LIN {X -0.181,Y -585.120,Z 1414.971,A 0.000,B 0.000,C 90.000,E1 30.797} C_DIS
LIN {X -0.267,Y -582.013,Z 1414.967,A 0.000,B 0.000,C 90.000,E1 30.001} C_DIS
LIN {X -0.018,Y -577.192,Z 1414.961,A 0.000,B 0.000,C 90.000,E1 28.899} C_DIS
LIN {X -0.191,Y -573.056,Z 1414.956,A 0.000,B 0.000,C 90.000,E1 28.103} C_DIS
LIN {X 0.092,Y -568.645,Z 1414.952,A 0.000,B 0.000,C 90.000,E1 27.257} C_DIS
LIN {X 0.067,Y -563.902,Z 1414.947,A 0.000,B 0.000,C 90.000,E1 26.437} C_DIS
LIN {X -0.163,Y -559.631,Z 1414.943,A 0.000,B 0.000,C 90.000,E1 25.771} C_DIS
LIN {X 0.221,Y -554.124,Z 1414.938,A 0.000,B 0.000,C 90.000,E1 24.899} C_DIS
LIN {X -0.222,Y -550.199,Z 1414.935,A 0.000,B 0.000,C 90.000,E1 24.387} C_DIS
LIN {X 0.061,Y -543.773,Z 1414.931,A 0.000,B 0.000,C 90.000,E1 23.515} C_DIS
LIN {X -0.088,Y -538.027,Z 1414.927,A 0.000,B 0.000,C 90.000,E1 22.823} C_DIS
LIN {X -0.189,Y -529.500,Z 1414.921,A 0.000,B 0.000,C 90.000,E1 21.844} C_DIS
LIN {X -0.178,Y -524.439,Z 1414.918,A 0.000,B 0.000,C 90.000,E1 21.280} C_DIS
LIN {X -0.246,Y -515.235,Z 1414.913,A 0.000,B 0.000,C 90.000,E1 20.301} C_DIS
LIN {X 0.169,Y -504.397,Z 1414.906,A 0.000,B 0.000,C 90.000,E1 19.141} C_DIS
LIN {X 0.226,Y -493.820,Z 1414.901,A 0.000,B 0.000,C 90.000,E1 18.055} C_DIS
LIN {X -0.129,Y -476.219,Z 1414.890,A 0.000,B 0.000,C 90.000,E1 16.260} C_DIS
LIN {X -0.019,Y -462.613,Z 1414.882,A 0.000,B 0.000,C 90.000,E1 14.773} C_DIS
LIN {X -0.025,Y -453.110,Z 1414.876,A 0.000,B 0.000,C 90.000,E1 13.716} C_DIS
LIN {X 0.077,Y -438.094,Z 1414.867,A 0.000,B 0.000,C 90.000,E1 12.007} C_DIS
LIN {X 0.034,Y -420.561,Z 1414.855,A 0.000,B 0.000,C 90.000,E1 9.905} C_DIS
LIN {X -0.065,Y -404.897,Z 1414.844,A 0.000,B 0.000,C 90.000,E1 7.871} C_DIS
LIN {X 0.079,Y -389.907,Z 1414.832,A 0.000,B 0.000,C 90.000,E1 5.796} C_DIS
LIN {X 0.032,Y -388.630,Z 1414.831,A 0.000,B 0.000,C 90.000,E1 5.625} C_DIS
LIN {X -0.056,Y -384.934,Z 1414.828,A 0.000,B 0.000,C 90.000,E1 4.992} C_DIS
LIN {X 0.034,Y -384.710,Z 1414.827,A 0.000,B 0.000,C 90.000,E1 4.878} C_DIS
LIN {X -0.003,Y -384.706,Z 1414.827,A 0.000,B 0.000,C 90.000,E1 4.878} C_DIS
LIN {X 0.112,Y -386.090,Z 1414.825,A 0.000,B 0.000,C 90.000,E1 4.473} C_DIS
LIN {X 0.057,Y -386.910,Z 1414.824,A 0.000,B 0.000,C 90.000,E1 4.302} C_DIS
LIN {X -0.075,Y -390.185,Z 1414.821,A 0.000,B 0.000,C 90.000,E1 3.784} C_DIS
LIN {X 0.181,Y -393.301,Z 1414.818,A 0.000,B 0.000,C 90.000,E1 3.212} C_DIS
LIN {X 0.160,Y -394.127,Z 1414.817,A 0.000,B 0.000,C 90.000,E1 3.037} C_DIS
LIN {X 0.084,Y -394.922,Z 1414.815,A 0.000,B 0.000,C 90.000,E1 2.694} C_DIS
LIN {X 0.145,Y -394.640,Z 1414.814,A 0.000,B 0.000,C 90.000,E1 2.579} C_DIS
LIN {X -0.179,Y -394.309,Z 1414.814,A 0.000,B 0.000,C 90.000,E1 2.579} C_DIS
LIN {X 0.177,Y -393.144,Z 1414.814,A 0.000,B 0.000,C 90.000,E1 2.465} C_DIS
LIN {X 0.102,Y -392.450,Z 1414.814,A 0.000,B 0.000,C 90.000,E1 2.465} C_DIS
LIN {X 0.060,Y -361.246,Z 1414.814,A 0.000,B 0.000,C 90.000,E1 2.465} C_DIS
LIN {X -0.064,Y -360.858,Z 1414.801,A 0.000,B 0.000,C 90.000,E1 0.115} C_DIS
LIN {X -0.053,Y -359.426,Z 1414.770,A 0.000,B 0.000,C 90.000,E1 354.546} C_DIS
LIN {X 0.070,Y -358.890,Z 1414.759,A 0.000,B 0.000,C 90.000,E1 352.648} C_DIS
LIN {X -0.020,Y -359.563,Z 1414.726,A 0.000,B 0.000,C 90.000,E1 346.645} C_DIS
LIN {X 0.001,Y -361.801,Z 1414.684,A 0.000,B 0.000,C 90.000,E1 339.135} C_DIS
LIN {X -0.154,Y -362.053,Z 1414.680,A 0.000,B 0.000,C 90.000,E1 338.411} C_DIS
LIN {X 0.189,Y -365.980,Z 1414.643,A 0.000,B 0.000,C 90.000,E1 331.641} C_DIS
LIN {X 0.029,Y -366.387,Z 1414.639,A 0.000,B 0.000,C 90.000,E1 330.923} C_DIS
LIN {X -0.031,Y -371.355,Z 1414.604,A 0.000,B 0.000,C 90.000,E1 324.642} C_DIS
LIN {X -0.043,Y -371.766,Z 1414.602,A 0.000,B 0.000,C 90.000,E1 324.276} C_DIS
LIN {X 0.013,Y -377.358,Z 1414.567,A 0.000,B 0.000,C 90.000,E1 318.038} C_DIS
LIN {X 0.012,Y -378.235,Z 1414.563,A 0.000,B 0.000,C 90.000,E1 317.310} C_DIS
LIN {X 0.002,Y -383.940,Z 1414.531,A 0.000,B 0.000,C 90.000,E1 311.515} C_DIS
LIN {X 0.088,Y -384.893,Z 1414.527,A 0.000,B 0.000,C 90.000,E1 310.782} C_DIS
LIN {X 0.262,Y -390.610,Z 1414.495,A 0.000,B 0.000,C 90.000,E1 305.025} C_DIS
LIN {X 0.106,Y -391.104,Z 1414.493,A 0.000,B 0.000,C 90.000,E1 304.692} C_DIS
LIN {X 0.022,Y -391.648,Z 1414.489,A 0.000,B 0.000,C 90.000,E1 303.992} C_DIS
LIN {X -0.080,Y -396.825,Z 1414.459,A 0.000,B 0.000,C 90.000,E1 298.693} C_DIS
LIN {X -0.210,Y -397.120,Z 1414.457,A 0.000,B 0.000,C 90.000,E1 298.359} C_DIS
LIN {X -0.055,Y -401.597,Z 1414.426,A 0.000,B 0.000,C 90.000,E1 292.717} C_DIS
LIN {X 0.222,Y -404.659,Z 1414.395,A 0.000,B 0.000,C 90.000,E1 287.094} C_DIS
LIN {X -0.079,Y -404.735,Z 1414.391,A 0.000,B 0.000,C 90.000,E1 286.441} C_DIS
LIN {X 0.214,Y -406.099,Z 1414.364,A 0.000,B 0.000,C 90.000,E1 281.535} C_DIS
LIN {X -0.176,Y -406.094,Z 1414.362,A 0.000,B 0.000,C 90.000,E1 281.243} C_DIS
LIN {X -0.097,Y -405.680,Z 1414.333,A 0.000,B 0.000,C 90.000,E1 276.024} C_DIS
LIN {X -0.165,Y -405.058,Z 1414.328,A 0.000,B 0.000,C 90.000,E1 274.992} C_DIS
LIN {X -0.060,Y -403.497,Z 1414.304,A 0.000,B 0.000,C 90.000,E1 270.802} C_DIS
LIN {X -0.092,Y -403.288,Z 1414.302,A 0.000,B 0.000,C 90.000,E1 270.458} C_DIS
LIN {X 0.091,Y -398.931,Z 1414.271,A 0.000,B 0.000,C 90.000,E1 264.837} C_DIS
LIN {X -0.040,Y -393.108,Z 1414.242,A 0.000,B 0.000,C 90.000,E1 259.567} C_DIS
LIN {X -0.079,Y -392.835,Z 1414.240,A 0.000,B 0.000,C 90.000,E1 259.218} C_DIS
LIN {X 0.034,Y -385.993,Z 1414.212,A 0.000,B 0.000,C 90.000,E1 254.212} C_DIS
LIN {X -0.026,Y -385.267,Z 1414.208,A 0.000,B 0.000,C 90.000,E1 253.504} C_DIS
LIN {X -0.004,Y -384.768,Z 1414.206,A 0.000,B 0.000,C 90.000,E1 253.142} C_DIS
LIN {X 0.221,Y -377.973,Z 1414.182,A 0.000,B 0.000,C 90.000,E1 248.773} C_DIS
LIN {X -0.044,Y -376.233,Z 1414.174,A 0.000,B 0.000,C 90.000,E1 247.358} C_DIS
LIN {X 0.057,Y -374.944,Z 1414.170,A 0.000,B 0.000,C 90.000,E1 246.613} C_DIS
LIN {X -0.208,Y -368.417,Z 1414.148,A 0.000,B 0.000,C 90.000,E1 242.615} C_DIS
LIN {X 0.097,Y -366.047,Z 1414.137,A 0.000,B 0.000,C 90.000,E1 240.717} C_DIS
LIN {X 0.004,Y -359.196,Z 1414.115,A 0.000,B 0.000,C 90.000,E1 236.628} C_DIS
LIN {X 0.021,Y -355.842,Z 1414.100,A 0.000,B 0.000,C 90.000,E1 233.989} C_DIS
LIN {X -0.173,Y -348.793,Z 1414.075,A 0.000,B 0.000,C 90.000,E1 229.461} C_DIS
LIN {X -0.097,Y -346.185,Z 1414.062,A 0.000,B 0.000,C 90.000,E1 227.148} C_DIS
LIN {X -0.088,Y -345.065,Z 1414.058,A 0.000,B 0.000,C 90.000,E1 226.377} C_DIS
LIN {X 0.094,Y -338.586,Z 1414.030,A 0.000,B 0.000,C 90.000,E1 221.310} C_DIS
LIN {X 0.094,Y -336.840,Z 1414.019,A 0.000,B 0.000,C 90.000,E1 219.358} C_DIS
LIN {X 0.014,Y -330.861,Z 1413.988,A 0.000,B 0.000,C 90.000,E1 213.865} C_DIS
LIN {X 0.149,Y -329.296,Z 1413.975,A 0.000,B 0.000,C 90.000,E1 211.465} C_DIS
LIN {X -0.154,Y -324.669,Z 1413.942,A 0.000,B 0.000,C 90.000,E1 205.540} C_DIS
LIN {X 0.174,Y -323.837,Z 1413.928,A 0.000,B 0.000,C 90.000,E1 203.078} C_DIS
LIN {X -0.017,Y -321.124,Z 1413.881,A 0.000,B 0.000,C 90.000,E1 194.662} C_DIS
LIN {X 0.138,Y -320.932,Z 1413.877,A 0.000,B 0.000,C 90.000,E1 193.828} C_DIS
LIN {X -0.076,Y -321.562,Z 1413.832,A 0.000,B 0.000,C 90.000,E1 185.796} C_DIS
LIN {X 0.028,Y -324.613,Z 1413.788,A 0.000,B 0.000,C 90.000,E1 177.879} C_DIS
LIN {X -0.001,Y -369.788,Z 1413.788,A 0.000,B 0.000,C 90.000,E1 177.879} C_DIS
LIN {X -0.100,Y -370.437,Z 1413.788,A 0.000,B 0.000,C 90.000,E1 177.879} C_DIS
LIN {X -0.163,Y -371.745,Z 1413.787,A 0.000,B 0.000,C 90.000,E1 177.764} C_DIS
LIN {X 0.129,Y -371.968,Z 1413.786,A 0.000,B 0.000,C 90.000,E1 177.421} C_DIS
LIN {X -0.028,Y -371.127,Z 1413.784,A 0.000,B 0.000,C 90.000,E1 177.078} C_DIS
LIN {X -0.164,Y -369.706,Z 1413.782,A 0.000,B 0.000,C 90.000,E1 176.731} C_DIS
LIN {X -0.043,Y -367.064,Z 1413.779,A 0.000,B 0.000,C 90.000,E1 176.159} C_DIS
LIN {X -0.167,Y -361.496,Z 1413.772,A 0.000,B 0.000,C 90.000,E1 175.065} C_DIS
LIN {X 0.067,Y -353.708,Z 1413.763,A 0.000,B 0.000,C 90.000,E1 173.337} C_DIS
LIN {X -0.012,Y -350.458,Z 1413.759,A 0.000,B 0.000,C 90.000,E1 172.591} C_DIS
LIN {X 0.052,Y -348.273,Z 1413.756,A 0.000,B 0.000,C 90.000,E1 172.008} C_DIS
LIN {X 0.057,Y -346.571,Z 1413.753,A 0.000,B 0.000,C 90.000,E1 171.432} C_DIS
LIN {X -0.155,Y -345.675,Z 1413.750,A 0.000,B 0.000,C 90.000,E1 171.084} C_DIS
LIN {X 0.105,Y -345.470,Z 1413.749,A 0.000,B 0.000,C 90.000,E1 170.849} C_DIS
LIN {X -0.176,Y -346.572,Z 1413.746,A 0.000,B 0.000,C 90.000,E1 170.387} C_DIS
LIN {X 0.147,Y -346.583,Z 1413.746,A 0.000,B 0.000,C 90.000,E1 170.330} C_DIS
LIN {X 0.138,Y -350.049,Z 1413.743,A 0.000,B 0.000,C 90.000,E1 169.690} C_DIS
LIN {X 0.139,Y -355.200,Z 1413.739,A 0.000,B 0.000,C 90.000,E1 168.926} C_DIS
LIN {X -0.057,Y -365.136,Z 1413.731,A 0.000,B 0.000,C 90.000,E1 167.645} C_DIS
LIN {X 0.109,Y -378.091,Z 1413.723,A 0.000,B 0.000,C 90.000,E1 166.061} C_DIS
LIN {X -0.133,Y -389.975,Z 1413.716,A 0.000,B 0.000,C 90.000,E1 164.810} C_DIS
LIN {X 0.023,Y -405.320,Z 1413.707,A 0.000,B 0.000,C 90.000,E1 163.323} C_DIS
LIN {X 0.023,Y -427.399,Z 1413.697,A 0.000,B 0.000,C 90.000,E1 161.456} C_DIS
LIN {X 0.187,Y -439.822,Z 1413.691,A 0.000,B 0.000,C 90.000,E1 160.423} C_DIS
LIN {X -0.100,Y -449.020,Z 1413.687,A 0.000,B 0.000,C 90.000,E1 159.699} C_DIS
LIN {X 0.245,Y -459.545,Z 1413.682,A 0.000,B 0.000,C 90.000,E1 158.773} C_DIS
LIN {X -0.114,Y -471.624,Z 1413.677,A 0.000,B 0.000,C 90.000,E1 157.794} C_DIS
LIN {X -0.067,Y -483.367,Z 1413.671,A 0.000,B 0.000,C 90.000,E1 156.741} C_DIS
LIN {X -0.200,Y -489.109,Z 1413.668,A 0.000,B 0.000,C 90.000,E1 156.230} C_DIS
LIN {X -0.133,Y -497.590,Z 1413.663,A 0.000,B 0.000,C 90.000,E1 155.409} C_DIS
LIN {X -0.134,Y -504.281,Z 1413.660,A 0.000,B 0.000,C 90.000,E1 154.717} C_DIS
LIN {X -0.177,Y -509.512,Z 1413.656,A 0.000,B 0.000,C 90.000,E1 154.152} C_DIS
LIN {X -0.115,Y -514.555,Z 1413.653,A 0.000,B 0.000,C 90.000,E1 153.563} C_DIS
LIN {X 0.122,Y -519.221,Z 1413.650,A 0.000,B 0.000,C 90.000,E1 152.948} C_DIS
LIN {X -0.140,Y -522.583,Z 1413.647,A 0.000,B 0.000,C 90.000,E1 152.538} C_DIS
LIN {X -0.072,Y -526.624,Z 1413.644,A 0.000,B 0.000,C 90.000,E1 151.948} C_DIS
LIN {X -0.225,Y -530.195,Z 1413.641,A 0.000,B 0.000,C 90.000,E1 151.385} C_DIS
LIN {X -0.102,Y -533.402,Z 1413.638,A 0.000,B 0.000,C 90.000,E1 150.795} C_DIS
LIN {X -0.097,Y -536.781,Z 1413.634,A 0.000,B 0.000,C 90.000,E1 150.078} C_DIS
LIN {X 0.209,Y -539.730,Z 1413.630,A 0.000,B 0.000,C 90.000,E1 149.331} C_DIS
LIN {X -0.064,Y -541.811,Z 1413.627,A 0.000,B 0.000,C 90.000,E1 148.791} C_DIS
LIN {X 0.141,Y -543.708,Z 1413.623,A 0.000,B 0.000,C 90.000,E1 148.201} C_DIS
LIN {X -0.077,Y -546.185,Z 1413.619,A 0.000,B 0.000,C 90.000,E1 147.375} C_DIS
LIN {X 0.193,Y -548.338,Z 1413.614,A 0.000,B 0.000,C 90.000,E1 146.501} C_DIS
LIN {X 0.025,Y -550.219,Z 1413.609,A 0.000,B 0.000,C 90.000,E1 145.674} C_DIS
LIN {X -0.126,Y -551.838,Z 1413.605,A 0.000,B 0.000,C 90.000,E1 144.848} C_DIS
LIN {X 0.057,Y -553.083,Z 1413.600,A 0.000,B 0.000,C 90.000,E1 143.989} C_DIS
LIN {X 0.330,Y -554.388,Z 1413.594,A 0.000,B 0.000,C 90.000,E1 142.844} C_DIS
LIN {X 0.258,Y -555.677,Z 1413.586,A 0.000,B 0.000,C 90.000,E1 141.457} C_DIS
LIN {X 0.206,Y -556.956,Z 1413.578,A 0.000,B 0.000,C 90.000,E1 140.070} C_DIS
LIN {X 0.029,Y -557.779,Z 1413.572,A 0.000,B 0.000,C 90.000,E1 138.976} C_DIS
LIN {X -0.084,Y -558.462,Z 1413.566,A 0.000,B 0.000,C 90.000,E1 137.877} C_DIS
LIN {X -0.118,Y -559.349,Z 1413.557,A 0.000,B 0.000,C 90.000,E1 136.215} C_DIS
LIN {X 0.261,Y -559.936,Z 1413.547,A 0.000,B 0.000,C 90.000,E1 134.514} C_DIS
LIN {X 0.263,Y -560.363,Z 1413.538,A 0.000,B 0.000,C 90.000,E1 132.852} C_DIS
LIN {X -0.109,Y -560.500,Z 1413.529,A 0.000,B 0.000,C 90.000,E1 131.229} C_DIS
LIN {X -0.061,Y -560.609,Z 1413.520,A 0.000,B 0.000,C 90.000,E1 129.564} C_DIS
LIN {X -0.027,Y -560.846,Z 1413.512,A 0.000,B 0.000,C 90.000,E1 128.177} C_DIS
LIN {X -0.088,Y -560.915,Z 1413.506,A 0.000,B 0.000,C 90.000,E1 127.076} C_DIS
LIN {X 0.160,Y -560.886,Z 1413.497,A 0.000,B 0.000,C 90.000,E1 125.391} C_DIS
LIN {X -0.371,Y -560.845,Z 1413.488,A 0.000,B 0.000,C 90.000,E1 123.785} C_DIS
LIN {X 0.155,Y -560.722,Z 1413.481,A 0.000,B 0.000,C 90.000,E1 122.625} C_DIS
LIN {X -0.218,Y -560.986,Z 1413.472,A 0.000,B 0.000,C 90.000,E1 121.003} C_DIS
LIN {X -0.084,Y -561.945,Z 1413.465,A 0.000,B 0.000,C 90.000,E1 119.745} C_DIS
LIN {X 0.093,Y -562.121,Z 1413.464,A 0.000,B 0.000,C 90.000,E1 119.589} C_DIS
LIN {X 0.000,Y -562.562,Z 1413.464,A 0.000,B 0.000,C 90.000,E1 119.461} C_DIS
LIN {X -0.185,Y -563.216,Z 1413.461,A 0.000,B 0.000,C 90.000,E1 118.949} C_DIS
LIN {X -0.227,Y -563.235,Z 1413.461,A 0.000,B 0.000,C 90.000,E1 118.949} C_DIS
LIN {X 0.271,Y -564.453,Z 1413.460,A 0.000,B 0.000,C 90.000,E1 118.743} C_DIS
LIN {X 0.026,Y -565.364,Z 1413.459,A 0.000,B 0.000,C 90.000,E1 118.615} C_DIS
LIN {X 0.248,Y -567.681,Z 1413.458,A 0.000,B 0.000,C 90.000,E1 118.487} C_DIS
LIN {X -0.019,Y -570.112,Z 1413.458,A 0.000,B 0.000,C 90.000,E1 118.437} C_DIS
LIN {X -0.161,Y -576.262,Z 1413.457,A 0.000,B 0.000,C 90.000,E1 118.281} C_DIS
LIN {X 0.030,Y -581.879,Z 1413.456,A 0.000,B 0.000,C 90.000,E1 118.025} C_DIS
LIN {X 0.230,Y -586.843,Z 1413.454,A 0.000,B 0.000,C 90.000,E1 117.641} C_DIS
LIN {X -0.142,Y -591.778,Z 1413.451,A 0.000,B 0.000,C 90.000,E1 117.206} C_DIS
LIN {X 0.057,Y -595.584,Z 1413.448,A 0.000,B 0.000,C 90.000,E1 116.668} C_DIS
LIN {X -0.124,Y -597.600,Z 1413.445,A 0.000,B 0.000,C 90.000,E1 116.155} C_DIS
LIN {X 0.329,Y -598.569,Z 1413.444,A 0.000,B 0.000,C 90.000,E1 115.848} C_DIS
LIN {X 0.248,Y -598.622,Z 1413.442,A 0.000,B 0.000,C 90.000,E1 115.591} C_DIS
LIN {X 0.169,Y -598.178,Z 1413.441,A 0.000,B 0.000,C 90.000,E1 115.335} C_DIS
LIN {X 0.092,Y -597.593,Z 1413.439,A 0.000,B 0.000,C 90.000,E1 115.079} C_DIS
LIN {X -0.072,Y -595.107,Z 1413.437,A 0.000,B 0.000,C 90.000,E1 114.567} C_DIS
LIN {X -0.363,Y -593.977,Z 1413.436,A 0.000,B 0.000,C 90.000,E1 114.463} C_DIS
LIN {X -0.008,Y -588.042,Z 1413.433,A 0.000,B 0.000,C 90.000,E1 113.951} C_DIS
LIN {X 0.118,Y -578.762,Z 1413.431,A 0.000,B 0.000,C 90.000,E1 113.515} C_DIS
LIN {X -0.216,Y -573.963,Z 1413.430,A 0.000,B 0.000,C 90.000,E1 113.334} C_DIS
LIN {X -0.131,Y -572.792,Z 1413.429,A 0.000,B 0.000,C 90.000,E1 113.259} C_DIS
LIN {X 0.165,Y -570.911,Z 1413.428,A 0.000,B 0.000,C 90.000,E1 113.078} C_DIS
LIN {X 0.129,Y -570.896,Z 1413.428,A 0.000,B 0.000,C 90.000,E1 113.078} C_DIS
LIN {X -0.056,Y -571.498,Z 1413.427,A 0.000,B 0.000,C 90.000,E1 112.823} C_DIS
LIN {X 0.130,Y -571.823,Z 1413.427,A 0.000,B 0.000,C 90.000,E1 112.770} C_DIS
LIN {X -0.294,Y -576.631,Z 1413.425,A 0.000,B 0.000,C 90.000,E1 112.461} C_DIS
LIN {X 0.149,Y -585.315,Z 1413.422,A 0.000,B 0.000,C 90.000,E1 111.972} C_DIS
LIN {X -0.035,Y -591.295,Z 1413.420,A 0.000,B 0.000,C 90.000,E1 111.642} C_DIS
LIN {X 0.186,Y -596.872,Z 1413.418,A 0.000,B 0.000,C 90.000,E1 111.227} C_DIS
LIN {X -0.342,Y -603.668,Z 1413.415,A 0.000,B 0.000,C 90.000,E1 110.737} C_DIS
LIN {X 0.063,Y -607.656,Z 1413.413,A 0.000,B 0.000,C 90.000,E1 110.355} C_DIS
LIN {X -0.126,Y -616.197,Z 1413.408,A 0.000,B 0.000,C 90.000,E1 109.504} C_DIS
LIN {X 0.233,Y -618.472,Z 1413.407,A 0.000,B 0.000,C 90.000,E1 109.214} C_DIS
LIN {X 0.230,Y -623.472,Z 1413.403,A 0.000,B 0.000,C 90.000,E1 108.598} C_DIS
LIN {X -0.217,Y -627.990,Z 1413.400,A 0.000,B 0.000,C 90.000,E1 108.000} C_DIS
LIN {X 0.166,Y -631.146,Z 1413.397,A 0.000,B 0.000,C 90.000,E1 107.457} C_DIS
LIN {X -0.033,Y -633.234,Z 1413.395,A 0.000,B 0.000,C 90.000,E1 107.094} C_DIS
LIN {X 0.202,Y -635.492,Z 1413.392,A 0.000,B 0.000,C 90.000,E1 106.567} C_DIS
LIN {X 0.202,Y -636.459,Z 1413.391,A 0.000,B 0.000,C 90.000,E1 106.315} C_DIS
LIN {X -0.321,Y -638.450,Z 1413.387,A 0.000,B 0.000,C 90.000,E1 105.607} C_DIS
LIN {X 0.127,Y -639.267,Z 1413.384,A 0.000,B 0.000,C 90.000,E1 105.064} C_DIS
LIN {X -0.069,Y -641.018,Z 1413.377,A 0.000,B 0.000,C 90.000,E1 103.828} C_DIS
LIN {X 0.238,Y -641.536,Z 1413.374,A 0.000,B 0.000,C 90.000,E1 103.300} C_DIS
LIN {X -0.234,Y -641.886,Z 1413.370,A 0.000,B 0.000,C 90.000,E1 102.591} C_DIS
LIN {X 0.079,Y -641.972,Z 1413.367,A 0.000,B 0.000,C 90.000,E1 102.063} C_DIS
LIN {X 0.232,Y -641.438,Z 1413.363,A 0.000,B 0.000,C 90.000,E1 101.299} C_DIS
LIN {X -0.211,Y -640.841,Z 1413.360,A 0.000,B 0.000,C 90.000,E1 100.838} C_DIS
LIN {X 0.093,Y -640.015,Z 1413.357,A 0.000,B 0.000,C 90.000,E1 100.310} C_DIS
LIN {X -0.353,Y -639.007,Z 1413.355,A 0.000,B 0.000,C 90.000,E1 99.849} C_DIS
LIN {X -0.064,Y -637.763,Z 1413.352,A 0.000,B 0.000,C 90.000,E1 99.321} C_DIS
LIN {X 0.111,Y -636.241,Z 1413.349,A 0.000,B 0.000,C 90.000,E1 98.803} C_DIS
LIN {X -0.257,Y -634.446,Z 1413.346,A 0.000,B 0.000,C 90.000,E1 98.333} C_DIS
LIN {X 0.243,Y -631.304,Z 1413.342,A 0.000,B 0.000,C 90.000,E1 97.530} C_DIS
LIN {X 0.315,Y -628.322,Z 1413.339,A 0.000,B 0.000,C 90.000,E1 96.891} C_DIS
LIN {X -0.195,Y -625.668,Z 1413.336,A 0.000,B 0.000,C 90.000,E1 96.429} C_DIS
LIN {X -0.026,Y -619.818,Z 1413.330,A 0.000,B 0.000,C 90.000,E1 95.391} C_DIS
LIN {X -0.131,Y -615.309,Z 1413.326,A 0.000,B 0.000,C 90.000,E1 94.759} C_DIS
LIN {X -0.157,Y -611.130,Z 1413.324,A 0.000,B 0.000,C 90.000,E1 94.245} C_DIS
LIN {X 0.095,Y -604.882,Z 1413.320,A 0.000,B 0.000,C 90.000,E1 93.612} C_DIS
LIN {X -0.180,Y -596.624,Z 1413.316,A 0.000,B 0.000,C 90.000,E1 92.922} C_DIS
LIN {X 0.039,Y -591.374,Z 1413.314,A 0.000,B 0.000,C 90.000,E1 92.465} C_DIS
LIN {X 0.127,Y -588.184,Z 1413.313,A 0.000,B 0.000,C 90.000,E1 92.236} C_DIS
LIN {X -0.110,Y -583.427,Z 1413.311,A 0.000,B 0.000,C 90.000,E1 91.949} C_DIS
LIN {X -0.120,Y -578.213,Z 1413.309,A 0.000,B 0.000,C 90.000,E1 91.661} C_DIS
LIN {X 0.148,Y -576.935,Z 1413.309,A 0.000,B 0.000,C 90.000,E1 91.547} C_DIS
LIN {X -0.117,Y -573.871,Z 1413.307,A 0.000,B 0.000,C 90.000,E1 91.318} C_DIS
LIN {X -0.154,Y -573.850,Z 1413.307,A 0.000,B 0.000,C 90.000,E1 91.318} C_DIS
LIN {X -0.038,Y -573.072,Z 1413.306,A 0.000,B 0.000,C 90.000,E1 91.088} C_DIS
LIN {X 0.104,Y -572.717,Z 1413.305,A 0.000,B 0.000,C 90.000,E1 90.802} C_DIS
LIN {X -0.125,Y -572.843,Z 1413.301,A 0.000,B 0.000,C 90.000,E1 90.229} C_DIS
LIN {X -0.278,Y -574.493,Z 1413.291,A 0.000,B 0.000,C 90.000,E1 88.339} C_DIS
LIN {X -0.105,Y -575.761,Z 1413.283,A 0.000,B 0.000,C 90.000,E1 86.963} C_DIS
LIN {X 0.239,Y -578.107,Z 1413.270,A 0.000,B 0.000,C 90.000,E1 84.489} C_DIS
LIN {X -0.057,Y -580.476,Z 1413.258,A 0.000,B 0.000,C 90.000,E1 82.356} C_DIS
LIN {X 0.182,Y -581.729,Z 1413.252,A 0.000,B 0.000,C 90.000,E1 81.254} C_DIS
LIN {X -0.099,Y -583.827,Z 1413.241,A 0.000,B 0.000,C 90.000,E1 79.398} C_DIS
LIN {X -0.037,Y -585.236,Z 1413.234,A 0.000,B 0.000,C 90.000,E1 78.049} C_DIS
LIN {X 0.054,Y -586.329,Z 1413.226,A 0.000,B 0.000,C 90.000,E1 76.700} C_DIS
LIN {X -0.095,Y -587.227,Z 1413.220,A 0.000,B 0.000,C 90.000,E1 75.644} C_DIS
LIN {X 0.159,Y -588.102,Z 1413.213,A 0.000,B 0.000,C 90.000,E1 74.283} C_DIS
LIN {X 0.025,Y -588.864,Z 1413.205,A 0.000,B 0.000,C 90.000,E1 72.960} C_DIS
LIN {X -0.090,Y -589.636,Z 1413.198,A 0.000,B 0.000,C 90.000,E1 71.638} C_DIS
LIN {X -0.215,Y -590.805,Z 1413.186,A 0.000,B 0.000,C 90.000,E1 69.518} C_DIS
LIN {X 0.210,Y -591.874,Z 1413.176,A 0.000,B 0.000,C 90.000,E1 67.614} C_DIS
LIN {X -0.200,Y -593.137,Z 1413.165,A 0.000,B 0.000,C 90.000,E1 65.793} C_DIS
LIN {X 0.212,Y -594.530,Z 1413.155,A 0.000,B 0.000,C 90.000,E1 63.896} C_DIS
LIN {X -0.238,Y -595.595,Z 1413.148,A 0.000,B 0.000,C 90.000,E1 62.615} C_DIS
LIN {X 0.042,Y -596.870,Z 1413.139,A 0.000,B 0.000,C 90.000,E1 61.001} C_DIS
LIN {X 0.202,Y -598.067,Z 1413.132,A 0.000,B 0.000,C 90.000,E1 59.665} C_DIS
LIN {X -0.121,Y -599.261,Z 1413.124,A 0.000,B 0.000,C 90.000,E1 58.377} C_DIS
LIN {X -0.002,Y -600.742,Z 1413.115,A 0.000,B 0.000,C 90.000,E1 56.786} C_DIS
LIN {X -0.297,Y -602.410,Z 1413.105,A 0.000,B 0.000,C 90.000,E1 54.975} C_DIS
LIN {X 0.027,Y -603.766,Z 1413.097,A 0.000,B 0.000,C 90.000,E1 53.371} C_DIS
LIN {X -0.225,Y -604.919,Z 1413.088,A 0.000,B 0.000,C 90.000,E1 51.823} C_DIS
LIN {X -0.238,Y -605.804,Z 1413.081,A 0.000,B 0.000,C 90.000,E1 50.517} C_DIS
LIN {X 0.142,Y -606.414,Z 1413.073,A 0.000,B 0.000,C 90.000,E1 49.175} C_DIS
LIN {X -0.187,Y -606.610,Z 1413.068,A 0.000,B 0.000,C 90.000,E1 48.162} C_DIS
LIN {X 0.220,Y -606.844,Z 1413.057,A 0.000,B 0.000,C 90.000,E1 46.296} C_DIS
LIN {X 0.321,Y -606.796,Z 1413.052,A 0.000,B 0.000,C 90.000,E1 45.243} C_DIS
LIN {X 0.233,Y -606.510,Z 1413.044,A 0.000,B 0.000,C 90.000,E1 43.947} C_DIS
LIN {X -0.091,Y -606.069,Z 1413.039,A 0.000,B 0.000,C 90.000,E1 42.933} C_DIS
LIN {X 0.239,Y -605.281,Z 1413.031,A 0.000,B 0.000,C 90.000,E1 41.595} C_DIS
LIN {X 0.349,Y -604.477,Z 1413.025,A 0.000,B 0.000,C 90.000,E1 40.539} C_DIS
LIN {X -0.148,Y -603.187,Z 1413.018,A 0.000,B 0.000,C 90.000,E1 39.277} C_DIS
LIN {X 0.147,Y -602.340,Z 1413.014,A 0.000,B 0.000,C 90.000,E1 38.463} C_DIS
LIN {X 0.330,Y -600.163,Z 1413.005,A 0.000,B 0.000,C 90.000,E1 36.870} C_DIS
LIN {X -0.019,Y -598.398,Z 1412.999,A 0.000,B 0.000,C 90.000,E1 35.851} C_DIS
LIN {X -0.028,Y -595.763,Z 1412.992,A 0.000,B 0.000,C 90.000,E1 34.532} C_DIS
LIN {X 0.309,Y -593.963,Z 1412.987,A 0.000,B 0.000,C 90.000,E1 33.706} C_DIS
LIN {X -0.099,Y -590.533,Z 1412.980,A 0.000,B 0.000,C 90.000,E1 32.418} C_DIS
LIN {X -0.014,Y -588.989,Z 1412.977,A 0.000,B 0.000,C 90.000,E1 31.878} C_DIS
LIN {X -0.059,Y -586.392,Z 1412.973,A 0.000,B 0.000,C 90.000,E1 31.082} C_DIS
LIN {X -0.003,Y -584.502,Z 1412.970,A 0.000,B 0.000,C 90.000,E1 30.541} C_DIS
LIN {X 0.038,Y -582.385,Z 1412.967,A 0.000,B 0.000,C 90.000,E1 30.001} C_DIS
LIN {X -0.077,Y -578.816,Z 1412.962,A 0.000,B 0.000,C 90.000,E1 29.205} C_DIS
LIN {X -0.084,Y -576.251,Z 1412.959,A 0.000,B 0.000,C 90.000,E1 28.665} C_DIS
LIN {X -0.040,Y -572.080,Z 1412.955,A 0.000,B 0.000,C 90.000,E1 27.847} C_DIS
LIN {X 0.231,Y -567.570,Z 1412.950,A 0.000,B 0.000,C 90.000,E1 27.001} C_DIS
LIN {X -0.217,Y -563.578,Z 1412.946,A 0.000,B 0.000,C 90.000,E1 26.360} C_DIS
LIN {X -0.190,Y -559.295,Z 1412.943,A 0.000,B 0.000,C 90.000,E1 25.668} C_DIS
LIN {X -0.070,Y -553.729,Z 1412.938,A 0.000,B 0.000,C 90.000,E1 24.823} C_DIS
LIN {X 0.097,Y -550.807,Z 1412.936,A 0.000,B 0.000,C 90.000,E1 24.387} C_DIS
LIN {X 0.259,Y -543.298,Z 1412.930,A 0.000,B 0.000,C 90.000,E1 23.387} C_DIS
LIN {X 0.100,Y -537.480,Z 1412.926,A 0.000,B 0.000,C 90.000,E1 22.695} C_DIS
LIN {X 0.183,Y -531.323,Z 1412.922,A 0.000,B 0.000,C 90.000,E1 21.972} C_DIS
LIN {X -0.044,Y -524.954,Z 1412.918,A 0.000,B 0.000,C 90.000,E1 21.280} C_DIS
LIN {X 0.219,Y -514.436,Z 1412.912,A 0.000,B 0.000,C 90.000,E1 20.120} C_DIS
LIN {X -0.002,Y -503.542,Z 1412.906,A 0.000,B 0.000,C 90.000,E1 19.033} C_DIS
LIN {X 0.056,Y -492.974,Z 1412.900,A 0.000,B 0.000,C 90.000,E1 17.946} C_DIS
LIN {X -0.092,Y -477.142,Z 1412.891,A 0.000,B 0.000,C 90.000,E1 16.315} C_DIS
LIN {X -0.167,Y -464.944,Z 1412.883,A 0.000,B 0.000,C 90.000,E1 15.009} C_DIS
LIN {X 0.017,Y -452.843,Z 1412.876,A 0.000,B 0.000,C 90.000,E1 13.647} C_DIS
LIN {X 0.219,Y -436.432,Z 1412.866,A 0.000,B 0.000,C 90.000,E1 11.771} C_DIS
LIN {X -0.023,Y -421.512,Z 1412.856,A 0.000,B 0.000,C 90.000,E1 10.018} C_DIS
LIN {X -0.114,Y -404.472,Z 1412.843,A 0.000,B 0.000,C 90.000,E1 7.814} C_DIS
LIN {X -0.062,Y -392.963,Z 1412.835,A 0.000,B 0.000,C 90.000,E1 6.258} C_DIS
LIN {X -0.148,Y -389.367,Z 1412.832,A 0.000,B 0.000,C 90.000,E1 5.739} C_DIS
LIN {X -0.061,Y -385.829,Z 1412.828,A 0.000,B 0.000,C 90.000,E1 5.049} C_DIS
LIN {X 0.060,Y -385.759,Z 1412.828,A 0.000,B 0.000,C 90.000,E1 4.992} C_DIS
LIN {X 0.023,Y -385.759,Z 1412.828,A 0.000,B 0.000,C 90.000,E1 4.992} C_DIS
LIN {X 0.029,Y -387.616,Z 1412.826,A 0.000,B 0.000,C 90.000,E1 4.588} C_DIS
LIN {X 0.096,Y -393.299,Z 1412.821,A 0.000,B 0.000,C 90.000,E1 3.841} C_DIS
LIN {X 0.100,Y -397.545,Z 1412.819,A 0.000,B 0.000,C 90.000,E1 3.326} C_DIS
LIN {X 0.053,Y -401.213,Z 1412.816,A 0.000,B 0.000,C 90.000,E1 2.808} C_DIS
LIN {X 0.025,Y -402.343,Z 1412.815,A 0.000,B 0.000,C 90.000,E1 2.636} C_DIS
LIN {X 0.003,Y -403.289,Z 1412.814,A 0.000,B 0.000,C 90.000,E1 2.465} C_DIS
LIN {X -0.018,Y -403.955,Z 1412.813,A 0.000,B 0.000,C 90.000,E1 2.293} C_DIS
LIN {X -0.053,Y -404.879,Z 1412.811,A 0.000,B 0.000,C 90.000,E1 1.949} C_DIS
LIN {X -0.072,Y -404.384,Z 1412.809,A 0.000,B 0.000,C 90.000,E1 1.604} C_DIS
LIN {X -0.133,Y -403.556,Z 1412.809,A 0.000,B 0.000,C 90.000,E1 1.547} C_DIS
LIN {X 0.115,Y -402.773,Z 1412.808,A 0.000,B 0.000,C 90.000,E1 1.489} C_DIS
LIN {X 0.090,Y -402.228,Z 1412.808,A 0.000,B 0.000,C 90.000,E1 1.489} C_DIS
LIN {X 0.057,Y -361.026,Z 1412.808,A 0.000,B 0.000,C 90.000,E1 1.489} C_DIS
LIN {X 0.000,Y -360.799,Z 1412.800,A 0.000,B 0.000,C 90.000,E1 360.000} C_DIS
LIN {X -0.053,Y -359.426,Z 1412.770,A 0.000,B 0.000,C 90.000,E1 354.546} C_DIS
LIN {X 0.070,Y -358.890,Z 1412.759,A 0.000,B 0.000,C 90.000,E1 352.648} C_DIS
LIN {X -0.020,Y -359.563,Z 1412.726,A 0.000,B 0.000,C 90.000,E1 346.645} C_DIS
LIN {X 0.001,Y -361.801,Z 1412.684,A 0.000,B 0.000,C 90.000,E1 339.135} C_DIS
LIN {X -0.154,Y -362.053,Z 1412.680,A 0.000,B 0.000,C 90.000,E1 338.411} C_DIS
LIN {X 0.189,Y -365.980,Z 1412.643,A 0.000,B 0.000,C 90.000,E1 331.641} C_DIS
LIN {X 0.029,Y -366.387,Z 1412.639,A 0.000,B 0.000,C 90.000,E1 330.923} C_DIS
LIN {X -0.031,Y -371.355,Z 1412.604,A 0.000,B 0.000,C 90.000,E1 324.642} C_DIS
LIN {X -0.043,Y -371.766,Z 1412.602,A 0.000,B 0.000,C 90.000,E1 324.276} C_DIS
LIN {X 0.013,Y -377.358,Z 1412.567,A 0.000,B 0.000,C 90.000,E1 318.038} C_DIS
LIN {X 0.012,Y -378.235,Z 1412.563,A 0.000,B 0.000,C 90.000,E1 317.310} C_DIS
LIN {X 0.002,Y -383.940,Z 1412.531,A 0.000,B 0.000,C 90.000,E1 311.515} C_DIS
LIN {X 0.088,Y -384.893,Z 1412.527,A 0.000,B 0.000,C 90.000,E1 310.782} C_DIS
LIN {X 0.262,Y -390.610,Z 1412.495,A 0.000,B 0.000,C 90.000,E1 305.025} C_DIS
LIN {X 0.106,Y -391.104,Z 1412.493,A 0.000,B 0.000,C 90.000,E1 304.692} C_DIS
LIN {X 0.022,Y -391.648,Z 1412.489,A 0.000,B 0.000,C 90.000,E1 303.992} C_DIS
LIN {X -0.080,Y -396.825,Z 1412.459,A 0.000,B 0.000,C 90.000,E1 298.693} C_DIS
LIN {X -0.210,Y -397.120,Z 1412.457,A 0.000,B 0.000,C 90.000,E1 298.359} C_DIS
LIN {X -0.055,Y -401.597,Z 1412.426,A 0.000,B 0.000,C 90.000,E1 292.717} C_DIS
LIN {X 0.222,Y -404.659,Z 1412.395,A 0.000,B 0.000,C 90.000,E1 287.094} C_DIS
LIN {X -0.079,Y -404.735,Z 1412.391,A 0.000,B 0.000,C 90.000,E1 286.441} C_DIS
LIN {X 0.214,Y -406.099,Z 1412.364,A 0.000,B 0.000,C 90.000,E1 281.535} C_DIS
LIN {X -0.176,Y -406.094,Z 1412.362,A 0.000,B 0.000,C 90.000,E1 281.243} C_DIS
LIN {X -0.097,Y -405.680,Z 1412.333,A 0.000,B 0.000,C 90.000,E1 276.024} C_DIS
LIN {X -0.165,Y -405.058,Z 1412.328,A 0.000,B 0.000,C 90.000,E1 274.992} C_DIS
LIN {X -0.060,Y -403.497,Z 1412.304,A 0.000,B 0.000,C 90.000,E1 270.802} C_DIS
LIN {X -0.092,Y -403.288,Z 1412.302,A 0.000,B 0.000,C 90.000,E1 270.458} C_DIS
LIN {X 0.091,Y -398.931,Z 1412.271,A 0.000,B 0.000,C 90.000,E1 264.837} C_DIS
LIN {X -0.040,Y -393.108,Z 1412.242,A 0.000,B 0.000,C 90.000,E1 259.567} C_DIS
LIN {X -0.079,Y -392.835,Z 1412.240,A 0.000,B 0.000,C 90.000,E1 259.218} C_DIS
LIN {X 0.034,Y -385.993,Z 1412.212,A 0.000,B 0.000,C 90.000,E1 254.212} C_DIS
LIN {X -0.026,Y -385.267,Z 1412.208,A 0.000,B 0.000,C 90.000,E1 253.504} C_DIS
LIN {X -0.004,Y -384.768,Z 1412.206,A 0.000,B 0.000,C 90.000,E1 253.142} C_DIS
LIN {X 0.221,Y -377.973,Z 1412.182,A 0.000,B 0.000,C 90.000,E1 248.773} C_DIS
LIN {X -0.044,Y -376.233,Z 1412.174,A 0.000,B 0.000,C 90.000,E1 247.358} C_DIS
LIN {X 0.057,Y -374.944,Z 1412.170,A 0.000,B 0.000,C 90.000,E1 246.613} C_DIS
LIN {X -0.208,Y -368.417,Z 1412.148,A 0.000,B 0.000,C 90.000,E1 242.615} C_DIS
LIN {X 0.097,Y -366.047,Z 1412.137,A 0.000,B 0.000,C 90.000,E1 240.717} C_DIS
LIN {X 0.004,Y -359.196,Z 1412.115,A 0.000,B 0.000,C 90.000,E1 236.628} C_DIS
LIN {X 0.021,Y -355.842,Z 1412.100,A 0.000,B 0.000,C 90.000,E1 233.989} C_DIS
LIN {X -0.173,Y -348.793,Z 1412.075,A 0.000,B 0.000,C 90.000,E1 229.461} C_DIS
LIN {X -0.097,Y -346.185,Z 1412.062,A 0.000,B 0.000,C 90.000,E1 227.148} C_DIS
LIN {X -0.088,Y -345.065,Z 1412.058,A 0.000,B 0.000,C 90.000,E1 226.377} C_DIS
LIN {X 0.094,Y -338.586,Z 1412.030,A 0.000,B 0.000,C 90.000,E1 221.310} C_DIS
LIN {X 0.094,Y -336.840,Z 1412.019,A 0.000,B 0.000,C 90.000,E1 219.358} C_DIS
LIN {X 0.014,Y -330.861,Z 1411.988,A 0.000,B 0.000,C 90.000,E1 213.865} C_DIS
LIN {X 0.149,Y -329.296,Z 1411.975,A 0.000,B 0.000,C 90.000,E1 211.465} C_DIS
LIN {X -0.154,Y -324.669,Z 1411.942,A 0.000,B 0.000,C 90.000,E1 205.540} C_DIS
LIN {X 0.174,Y -323.837,Z 1411.928,A 0.000,B 0.000,C 90.000,E1 203.078} C_DIS
LIN {X -0.017,Y -321.124,Z 1411.881,A 0.000,B 0.000,C 90.000,E1 194.662} C_DIS
LIN {X 0.138,Y -320.932,Z 1411.877,A 0.000,B 0.000,C 90.000,E1 193.828} C_DIS
LIN {X -0.076,Y -321.562,Z 1411.832,A 0.000,B 0.000,C 90.000,E1 185.796} C_DIS
LIN {X -0.076,Y -323.867,Z 1411.794,A 0.000,B 0.000,C 90.000,E1 178.912} C_DIS
LIN {X -0.112,Y -378.063,Z 1411.794,A 0.000,B 0.000,C 90.000,E1 178.912} C_DIS
LIN {X 0.054,Y -379.375,Z 1411.794,A 0.000,B 0.000,C 90.000,E1 178.854} C_DIS
LIN {X -0.177,Y -380.724,Z 1411.792,A 0.000,B 0.000,C 90.000,E1 178.568} C_DIS
LIN {X 0.087,Y -380.146,Z 1411.790,A 0.000,B 0.000,C 90.000,E1 178.165} C_DIS
LIN {X -0.035,Y -378.922,Z 1411.788,A 0.000,B 0.000,C 90.000,E1 177.822} C_DIS
LIN {X -0.158,Y -377.378,Z 1411.786,A 0.000,B 0.000,C 90.000,E1 177.478} C_DIS
LIN {X -0.182,Y -371.549,Z 1411.780,A 0.000,B 0.000,C 90.000,E1 176.388} C_DIS
LIN {X -0.024,Y -368.480,Z 1411.777,A 0.000,B 0.000,C 90.000,E1 175.812} C_DIS
LIN {X -0.159,Y -362.873,Z 1411.771,A 0.000,B 0.000,C 90.000,E1 174.723} C_DIS
LIN {X 0.185,Y -352.562,Z 1411.758,A 0.000,B 0.000,C 90.000,E1 172.413} C_DIS
LIN {X 0.016,Y -349.061,Z 1411.753,A 0.000,B 0.000,C 90.000,E1 171.489} C_DIS
LIN {X 0.155,Y -348.083,Z 1411.751,A 0.000,B 0.000,C 90.000,E1 171.084} C_DIS
LIN {X -0.137,Y -347.027,Z 1411.748,A 0.000,B 0.000,C 90.000,E1 170.622} C_DIS
LIN {X -0.156,Y -347.026,Z 1411.748,A 0.000,B 0.000,C 90.000,E1 170.622} C_DIS
LIN {X 0.139,Y -347.488,Z 1411.746,A 0.000,B 0.000,C 90.000,E1 170.274} C_DIS
LIN {X 0.121,Y -347.495,Z 1411.746,A 0.000,B 0.000,C 90.000,E1 170.274} C_DIS
LIN {X 0.020,Y -351.133,Z 1411.742,A 0.000,B 0.000,C 90.000,E1 169.577} C_DIS
LIN {X -0.081,Y -356.382,Z 1411.738,A 0.000,B 0.000,C 90.000,E1 168.814} C_DIS
LIN {X -0.079,Y -363.392,Z 1411.733,A 0.000,B 0.000,C 90.000,E1 167.881} C_DIS
LIN {X -0.013,Y -376.468,Z 1411.724,A 0.000,B 0.000,C 90.000,E1 166.284} C_DIS
LIN {X -0.052,Y -388.281,Z 1411.717,A 0.000,B 0.000,C 90.000,E1 164.991} C_DIS
LIN {X -0.083,Y -400.479,Z 1411.710,A 0.000,B 0.000,C 90.000,E1 163.795} C_DIS
LIN {X 0.142,Y -420.789,Z 1411.700,A 0.000,B 0.000,C 90.000,E1 162.000} C_DIS
LIN {X 0.195,Y -431.760,Z 1411.695,A 0.000,B 0.000,C 90.000,E1 161.094} C_DIS
LIN {X -0.080,Y -441.171,Z 1411.691,A 0.000,B 0.000,C 90.000,E1 160.369} C_DIS
LIN {X 0.146,Y -452.033,Z 1411.686,A 0.000,B 0.000,C 90.000,E1 159.444} C_DIS
LIN {X -0.216,Y -462.681,Z 1411.681,A 0.000,B 0.000,C 90.000,E1 158.592} C_DIS
LIN {X 0.038,Y -471.698,Z 1411.677,A 0.000,B 0.000,C 90.000,E1 157.794} C_DIS
LIN {X 0.089,Y -483.431,Z 1411.671,A 0.000,B 0.000,C 90.000,E1 156.741} C_DIS
LIN {X -0.042,Y -489.177,Z 1411.668,A 0.000,B 0.000,C 90.000,E1 156.230} C_DIS
LIN {X 0.053,Y -497.629,Z 1411.663,A 0.000,B 0.000,C 90.000,E1 155.409} C_DIS
LIN {X 0.023,Y -504.327,Z 1411.660,A 0.000,B 0.000,C 90.000,E1 154.717} C_DIS
LIN {X -0.040,Y -509.583,Z 1411.656,A 0.000,B 0.000,C 90.000,E1 154.152} C_DIS
LIN {X -0.084,Y -513.462,Z 1411.654,A 0.000,B 0.000,C 90.000,E1 153.717} C_DIS
LIN {X 0.056,Y -520.480,Z 1411.649,A 0.000,B 0.000,C 90.000,E1 152.820} C_DIS
LIN {X -0.199,Y -523.742,Z 1411.647,A 0.000,B 0.000,C 90.000,E1 152.410} C_DIS
LIN {X -0.213,Y -526.777,Z 1411.644,A 0.000,B 0.000,C 90.000,E1 151.975} C_DIS
LIN {X -0.117,Y -530.348,Z 1411.641,A 0.000,B 0.000,C 90.000,E1 151.385} C_DIS
LIN {X 0.008,Y -533.556,Z 1411.638,A 0.000,B 0.000,C 90.000,E1 150.795} C_DIS
LIN {X 0.014,Y -536.935,Z 1411.634,A 0.000,B 0.000,C 90.000,E1 150.078} C_DIS
LIN {X -0.278,Y -539.339,Z 1411.631,A 0.000,B 0.000,C 90.000,E1 149.537} C_DIS
LIN {X -0.091,Y -541.441,Z 1411.627,A 0.000,B 0.000,C 90.000,E1 148.948} C_DIS
LIN {X 0.124,Y -544.247,Z 1411.623,A 0.000,B 0.000,C 90.000,E1 148.074} C_DIS
LIN {X -0.118,Y -545.934,Z 1411.620,A 0.000,B 0.000,C 90.000,E1 147.533} C_DIS
LIN {X -0.315,Y -548.127,Z 1411.615,A 0.000,B 0.000,C 90.000,E1 146.707} C_DIS
LIN {X 0.277,Y -550.021,Z 1411.610,A 0.000,B 0.000,C 90.000,E1 145.801} C_DIS
LIN {X 0.128,Y -551.641,Z 1411.606,A 0.000,B 0.000,C 90.000,E1 144.975} C_DIS
LIN {X -0.012,Y -552.924,Z 1411.601,A 0.000,B 0.000,C 90.000,E1 144.149} C_DIS
LIN {X -0.259,Y -553.972,Z 1411.596,A 0.000,B 0.000,C 90.000,E1 143.336} C_DIS
LIN {X 0.027,Y -555.036,Z 1411.590,A 0.000,B 0.000,C 90.000,E1 142.190} C_DIS
LIN {X 0.041,Y -556.570,Z 1411.581,A 0.000,B 0.000,C 90.000,E1 140.517} C_DIS
LIN {X 0.279,Y -557.462,Z 1411.575,A 0.000,B 0.000,C 90.000,E1 139.380} C_DIS
LIN {X -0.257,Y -558.167,Z 1411.568,A 0.000,B 0.000,C 90.000,E1 138.324} C_DIS
LIN {X -0.221,Y -559.213,Z 1411.558,A 0.000,B 0.000,C 90.000,E1 136.377} C_DIS
LIN {X -0.305,Y -559.684,Z 1411.550,A 0.000,B 0.000,C 90.000,E1 135.000} C_DIS
LIN {X 0.024,Y -560.132,Z 1411.542,A 0.000,B 0.000,C 90.000,E1 133.581} C_DIS
LIN {X 0.282,Y -560.342,Z 1411.536,A 0.000,B 0.000,C 90.000,E1 132.447} C_DIS
LIN {X -0.098,Y -560.453,Z 1411.527,A 0.000,B 0.000,C 90.000,E1 130.825} C_DIS
LIN {X -0.322,Y -560.672,Z 1411.516,A 0.000,B 0.000,C 90.000,E1 128.910} C_DIS
LIN {X -0.284,Y -560.879,Z 1411.508,A 0.000,B 0.000,C 90.000,E1 127.523} C_DIS
LIN {X 0.199,Y -560.867,Z 1411.501,A 0.000,B 0.000,C 90.000,E1 126.091} C_DIS
LIN {X -0.014,Y -560.850,Z 1411.491,A 0.000,B 0.000,C 90.000,E1 124.452} C_DIS
LIN {X -0.093,Y -560.779,Z 1411.482,A 0.000,B 0.000,C 90.000,E1 122.801} C_DIS
LIN {X -0.081,Y -561.040,Z 1411.474,A 0.000,B 0.000,C 90.000,E1 121.416} C_DIS
LIN {X 0.004,Y -561.167,Z 1411.473,A 0.000,B 0.000,C 90.000,E1 121.131} C_DIS
LIN {X 0.140,Y -562.433,Z 1411.466,A 0.000,B 0.000,C 90.000,E1 119.873} C_DIS
LIN {X 0.040,Y -562.756,Z 1411.465,A 0.000,B 0.000,C 90.000,E1 119.745} C_DIS
LIN {X -0.137,Y -564.201,Z 1411.463,A 0.000,B 0.000,C 90.000,E1 119.333} C_DIS
LIN {X -0.180,Y -564.221,Z 1411.463,A 0.000,B 0.000,C 90.000,E1 119.333} C_DIS
LIN {X -0.196,Y -564.906,Z 1411.463,A 0.000,B 0.000,C 90.000,E1 119.283} C_DIS
LIN {X -0.108,Y -566.280,Z 1411.462,A 0.000,B 0.000,C 90.000,E1 119.205} C_DIS
LIN {X -0.019,Y -568.317,Z 1411.462,A 0.000,B 0.000,C 90.000,E1 119.127} C_DIS
LIN {X 0.251,Y -574.394,Z 1411.461,A 0.000,B 0.000,C 90.000,E1 118.949} C_DIS
LIN {X 0.179,Y -578.503,Z 1411.461,A 0.000,B 0.000,C 90.000,E1 118.871} C_DIS
LIN {X -0.223,Y -583.864,Z 1411.459,A 0.000,B 0.000,C 90.000,E1 118.693} C_DIS
LIN {X -0.044,Y -586.053,Z 1411.459,A 0.000,B 0.000,C 90.000,E1 118.537} C_DIS
LIN {X -0.007,Y -590.143,Z 1411.457,A 0.000,B 0.000,C 90.000,E1 118.231} C_DIS
LIN {X -0.130,Y -595.170,Z 1411.454,A 0.000,B 0.000,C 90.000,E1 117.769} C_DIS
LIN {X -0.169,Y -598.702,Z 1411.452,A 0.000,B 0.000,C 90.000,E1 117.385} C_DIS
LIN {X -0.205,Y -599.778,Z 1411.451,A 0.000,B 0.000,C 90.000,E1 117.257} C_DIS
LIN {X -0.243,Y -600.652,Z 1411.451,A 0.000,B 0.000,C 90.000,E1 117.129} C_DIS
LIN {X 0.187,Y -602.791,Z 1411.448,A 0.000,B 0.000,C 90.000,E1 116.693} C_DIS
LIN {X 0.154,Y -603.387,Z 1411.448,A 0.000,B 0.000,C 90.000,E1 116.565} C_DIS
LIN {X 0.092,Y -604.334,Z 1411.446,A 0.000,B 0.000,C 90.000,E1 116.309} C_DIS
LIN {X 0.032,Y -604.851,Z 1411.445,A 0.000,B 0.000,C 90.000,E1 116.052} C_DIS
LIN {X -0.081,Y -605.335,Z 1411.442,A 0.000,B 0.000,C 90.000,E1 115.540} C_DIS
LIN {X -0.136,Y -604.566,Z 1411.440,A 0.000,B 0.000,C 90.000,E1 115.283} C_DIS
LIN {X -0.220,Y -603.124,Z 1411.438,A 0.000,B 0.000,C 90.000,E1 114.899} C_DIS
LIN {X 0.200,Y -599.397,Z 1411.435,A 0.000,B 0.000,C 90.000,E1 114.335} C_DIS
LIN {X 0.164,Y -598.119,Z 1411.435,A 0.000,B 0.000,C 90.000,E1 114.207} C_DIS
LIN {X 0.353,Y -593.033,Z 1411.433,A 0.000,B 0.000,C 90.000,E1 113.823} C_DIS
LIN {X -0.212,Y -591.314,Z 1411.432,A 0.000,B 0.000,C 90.000,E1 113.770} C_DIS
LIN {X -0.012,Y -581.869,Z 1411.430,A 0.000,B 0.000,C 90.000,E1 113.334} C_DIS
LIN {X -0.148,Y -576.718,Z 1411.428,A 0.000,B 0.000,C 90.000,E1 113.131} C_DIS
LIN {X -0.054,Y -574.072,Z 1411.427,A 0.000,B 0.000,C 90.000,E1 112.950} C_DIS
LIN {X -0.094,Y -574.076,Z 1411.427,A 0.000,B 0.000,C 90.000,E1 112.950} C_DIS
LIN {X 0.064,Y -575.335,Z 1411.427,A 0.000,B 0.000,C 90.000,E1 112.770} C_DIS
LIN {X -0.088,Y -576.059,Z 1411.426,A 0.000,B 0.000,C 90.000,E1 112.717} C_DIS
LIN {X -0.170,Y -578.168,Z 1411.425,A 0.000,B 0.000,C 90.000,E1 112.589} C_DIS
LIN {X 0.003,Y -587.306,Z 1411.423,A 0.000,B 0.000,C 90.000,E1 112.078} C_DIS
LIN {X 0.003,Y -593.235,Z 1411.421,A 0.000,B 0.000,C 90.000,E1 111.716} C_DIS
LIN {X -0.151,Y -598.889,Z 1411.418,A 0.000,B 0.000,C 90.000,E1 111.334} C_DIS
LIN {X 0.137,Y -604.351,Z 1411.416,A 0.000,B 0.000,C 90.000,E1 110.865} C_DIS
LIN {X -0.259,Y -608.408,Z 1411.414,A 0.000,B 0.000,C 90.000,E1 110.556} C_DIS
LIN {X -0.217,Y -613.387,Z 1411.411,A 0.000,B 0.000,C 90.000,E1 110.066} C_DIS
LIN {X 0.160,Y -619.420,Z 1411.408,A 0.000,B 0.000,C 90.000,E1 109.396} C_DIS
LIN {X -0.116,Y -624.576,Z 1411.404,A 0.000,B 0.000,C 90.000,E1 108.779} C_DIS
LIN {X 0.242,Y -628.336,Z 1411.401,A 0.000,B 0.000,C 90.000,E1 108.236} C_DIS
LIN {X -0.168,Y -632.485,Z 1411.398,A 0.000,B 0.000,C 90.000,E1 107.638} C_DIS
LIN {X 0.064,Y -635.834,Z 1411.394,A 0.000,B 0.000,C 90.000,E1 106.985} C_DIS
LIN {X -0.106,Y -638.295,Z 1411.391,A 0.000,B 0.000,C 90.000,E1 106.370} C_DIS
LIN {X 0.166,Y -639.755,Z 1411.388,A 0.000,B 0.000,C 90.000,E1 105.843} C_DIS
LIN {X 0.001,Y -640.405,Z 1411.387,A 0.000,B 0.000,C 90.000,E1 105.607} C_DIS
LIN {X -0.012,Y -642.221,Z 1411.380,A 0.000,B 0.000,C 90.000,E1 104.356} C_DIS
LIN {X 0.146,Y -643.138,Z 1411.376,A 0.000,B 0.000,C 90.000,E1 103.592} C_DIS
LIN {X -0.159,Y -643.584,Z 1411.373,A 0.000,B 0.000,C 90.000,E1 103.119} C_DIS
LIN {X 0.015,Y -643.826,Z 1411.369,A 0.000,B 0.000,C 90.000,E1 102.355} C_DIS
LIN {X -0.137,Y -643.858,Z 1411.367,A 0.000,B 0.000,C 90.000,E1 102.119} C_DIS
LIN {X -0.092,Y -643.301,Z 1411.363,A 0.000,B 0.000,C 90.000,E1 101.366} C_DIS
LIN {X 0.232,Y -642.742,Z 1411.360,A 0.000,B 0.000,C 90.000,E1 100.838} C_DIS
LIN {X -0.083,Y -641.940,Z 1411.358,A 0.000,B 0.000,C 90.000,E1 100.366} C_DIS
LIN {X 0.115,Y -640.934,Z 1411.355,A 0.000,B 0.000,C 90.000,E1 99.849} C_DIS
LIN {X 0.142,Y -638.959,Z 1411.351,A 0.000,B 0.000,C 90.000,E1 99.095} C_DIS
LIN {X -0.205,Y -637.388,Z 1411.348,A 0.000,B 0.000,C 90.000,E1 98.624} C_DIS
LIN {X -0.030,Y -635.578,Z 1411.345,A 0.000,B 0.000,C 90.000,E1 98.106} C_DIS
LIN {X -0.058,Y -632.208,Z 1411.341,A 0.000,B 0.000,C 90.000,E1 97.352} C_DIS
LIN {X 0.085,Y -629.790,Z 1411.338,A 0.000,B 0.000,C 90.000,E1 96.834} C_DIS
LIN {X 0.208,Y -627.150,Z 1411.335,A 0.000,B 0.000,C 90.000,E1 96.315} C_DIS
LIN {X 0.165,Y -623.512,Z 1411.332,A 0.000,B 0.000,C 90.000,E1 95.682} C_DIS
LIN {X -0.223,Y -621.238,Z 1411.330,A 0.000,B 0.000,C 90.000,E1 95.334} C_DIS
LIN {X -0.212,Y -617.795,Z 1411.327,A 0.000,B 0.000,C 90.000,E1 94.821} C_DIS
LIN {X 0.282,Y -612.567,Z 1411.323,A 0.000,B 0.000,C 90.000,E1 94.131} C_DIS
LIN {X -0.216,Y -606.176,Z 1411.320,A 0.000,B 0.000,C 90.000,E1 93.555} C_DIS
LIN {X -0.233,Y -598.237,Z 1411.316,A 0.000,B 0.000,C 90.000,E1 92.865} C_DIS
LIN {X -0.185,Y -591.262,Z 1411.313,A 0.000,B 0.000,C 90.000,E1 92.293} C_DIS
LIN {X -0.120,Y -588.016,Z 1411.311,A 0.000,B 0.000,C 90.000,E1 92.064} C_DIS
LIN {X -0.276,Y -583.239,Z 1411.310,A 0.000,B 0.000,C 90.000,E1 91.776} C_DIS
LIN {X -0.217,Y -578.127,Z 1411.308,A 0.000,B 0.000,C 90.000,E1 91.489} C_DIS
LIN {X 0.059,Y -575.438,Z 1411.307,A 0.000,B 0.000,C 90.000,E1 91.260} C_DIS
LIN {X 0.263,Y -573.829,Z 1411.306,A 0.000,B 0.000,C 90.000,E1 91.088} C_DIS
LIN {X 0.209,Y -573.787,Z 1411.306,A 0.000,B 0.000,C 90.000,E1 91.088} C_DIS
LIN {X -0.169,Y -573.239,Z 1411.305,A 0.000,B 0.000,C 90.000,E1 90.974} C_DIS
LIN {X -0.256,Y -572.841,Z 1411.304,A 0.000,B 0.000,C 90.000,E1 90.688} C_DIS
LIN {X 0.026,Y -572.915,Z 1411.301,A 0.000,B 0.000,C 90.000,E1 90.115} C_DIS
LIN {X -0.125,Y -574.575,Z 1411.290,A 0.000,B 0.000,C 90.000,E1 88.224} C_DIS
LIN {X 0.080,Y -575.821,Z 1411.283,A 0.000,B 0.000,C 90.000,E1 86.846} C_DIS
LIN {X -0.182,Y -578.175,Z 1411.269,A 0.000,B 0.000,C 90.000,E1 84.432} C_DIS
LIN {X -0.049,Y -580.269,Z 1411.259,A 0.000,B 0.000,C 90.000,E1 82.527} C_DIS
LIN {X -0.012,Y -582.140,Z 1411.250,A 0.000,B 0.000,C 90.000,E1 80.905} C_DIS
LIN {X 0.047,Y -583.965,Z 1411.241,A 0.000,B 0.000,C 90.000,E1 79.285} C_DIS
LIN {X 0.108,Y -585.329,Z 1411.233,A 0.000,B 0.000,C 90.000,E1 77.937} C_DIS
LIN {X 0.194,Y -586.404,Z 1411.226,A 0.000,B 0.000,C 90.000,E1 76.589} C_DIS
LIN {X 0.188,Y -587.315,Z 1411.220,A 0.000,B 0.000,C 90.000,E1 75.519} C_DIS
LIN {X -0.117,Y -588.181,Z 1411.212,A 0.000,B 0.000,C 90.000,E1 74.212} C_DIS
LIN {X 0.004,Y -589.065,Z 1411.203,A 0.000,B 0.000,C 90.000,E1 72.598} C_DIS
LIN {X -0.106,Y -589.822,Z 1411.196,A 0.000,B 0.000,C 90.000,E1 71.275} C_DIS
LIN {X 0.096,Y -590.853,Z 1411.186,A 0.000,B 0.000,C 90.000,E1 69.390} C_DIS
LIN {X -0.019,Y -591.967,Z 1411.175,A 0.000,B 0.000,C 90.000,E1 67.539} C_DIS
LIN {X 0.124,Y -593.222,Z 1411.165,A 0.000,B 0.000,C 90.000,E1 65.665} C_DIS
LIN {X 0.006,Y -594.636,Z 1411.155,A 0.000,B 0.000,C 90.000,E1 63.819} C_DIS
LIN {X 0.092,Y -595.697,Z 1411.147,A 0.000,B 0.000,C 90.000,E1 62.487} C_DIS
LIN {X -0.062,Y -596.775,Z 1411.140,A 0.000,B 0.000,C 90.000,E1 61.179} C_DIS
LIN {X -0.198,Y -597.967,Z 1411.133,A 0.000,B 0.000,C 90.000,E1 59.871} C_DIS
LIN {X -0.101,Y -599.430,Z 1411.124,A 0.000,B 0.000,C 90.000,E1 58.280} C_DIS
LIN {X -0.171,Y -600.865,Z 1411.115,A 0.000,B 0.000,C 90.000,E1 56.707} C_DIS
LIN {X 0.034,Y -602.548,Z 1411.105,A 0.000,B 0.000,C 90.000,E1 54.848} C_DIS
LIN {X -0.127,Y -603.907,Z 1411.096,A 0.000,B 0.000,C 90.000,E1 53.290} C_DIS
LIN {X -0.159,Y -604.867,Z 1411.089,A 0.000,B 0.000,C 90.000,E1 51.984} C_DIS
LIN {X -0.056,Y -605.585,Z 1411.083,A 0.000,B 0.000,C 90.000,E1 50.928} C_DIS
LIN {X -0.061,Y -606.290,Z 1411.076,A 0.000,B 0.000,C 90.000,E1 49.622} C_DIS
LIN {X -0.197,Y -606.568,Z 1411.071,A 0.000,B 0.000,C 90.000,E1 48.852} C_DIS
LIN {X -0.069,Y -606.730,Z 1411.066,A 0.000,B 0.000,C 90.000,E1 47.796} C_DIS
LIN {X -0.106,Y -606.937,Z 1411.055,A 0.000,B 0.000,C 90.000,E1 45.972} C_DIS
LIN {X -0.002,Y -606.819,Z 1411.050,A 0.000,B 0.000,C 90.000,E1 44.919} C_DIS
LIN {X -0.092,Y -606.466,Z 1411.042,A 0.000,B 0.000,C 90.000,E1 43.623} C_DIS
LIN {X 0.029,Y -605.978,Z 1411.036,A 0.000,B 0.000,C 90.000,E1 42.567} C_DIS
LIN {X -0.095,Y -605.161,Z 1411.029,A 0.000,B 0.000,C 90.000,E1 41.272} C_DIS
LIN {X 0.264,Y -603.989,Z 1411.022,A 0.000,B 0.000,C 90.000,E1 39.930} C_DIS
LIN {X -0.243,Y -602.657,Z 1411.015,A 0.000,B 0.000,C 90.000,E1 38.669} C_DIS
LIN {X -0.077,Y -601.274,Z 1411.009,A 0.000,B 0.000,C 90.000,E1 37.604} C_DIS
LIN {X 0.192,Y -600.172,Z 1411.005,A 0.000,B 0.000,C 90.000,E1 36.790} C_DIS
LIN {X 0.086,Y -598.861,Z 1411.000,A 0.000,B 0.000,C 90.000,E1 36.011} C_DIS
LIN {X 0.199,Y -596.836,Z 1410.994,A 0.000,B 0.000,C 90.000,E1 34.945} C_DIS
LIN {X -0.281,Y -595.166,Z 1410.990,A 0.000,B 0.000,C 90.000,E1 34.199} C_DIS
LIN {X 0.267,Y -592.607,Z 1410.984,A 0.000,B 0.000,C 90.000,E1 33.086} C_DIS
LIN {X -0.248,Y -590.466,Z 1410.980,A 0.000,B 0.000,C 90.000,E1 32.339} C_DIS
LIN {X -0.281,Y -588.073,Z 1410.975,A 0.000,B 0.000,C 90.000,E1 31.544} C_DIS
LIN {X -0.033,Y -585.400,Z 1410.971,A 0.000,B 0.000,C 90.000,E1 30.718} C_DIS
LIN {X -0.119,Y -582.219,Z 1410.966,A 0.000,B 0.000,C 90.000,E1 29.922} C_DIS
LIN {X 0.268,Y -578.646,Z 1410.962,A 0.000,B 0.000,C 90.000,E1 29.077} C_DIS
LIN {X -0.016,Y -576.056,Z 1410.959,A 0.000,B 0.000,C 90.000,E1 28.565} C_DIS
LIN {X -0.205,Y -571.859,Z 1410.954,A 0.000,B 0.000,C 90.000,E1 27.769} C_DIS
LIN {X -0.112,Y -568.094,Z 1410.950,A 0.000,B 0.000,C 90.000,E1 27.078} C_DIS
LIN {X 0.207,Y -564.138,Z 1410.947,A 0.000,B 0.000,C 90.000,E1 26.360} C_DIS
LIN {X -0.171,Y -560.751,Z 1410.944,A 0.000,B 0.000,C 90.000,E1 25.848} C_DIS
LIN {X -0.169,Y -556.249,Z 1410.940,A 0.000,B 0.000,C 90.000,E1 25.155} C_DIS
LIN {X -0.203,Y -551.471,Z 1410.936,A 0.000,B 0.000,C 90.000,E1 24.463} C_DIS
LIN {X 0.098,Y -545.060,Z 1410.931,A 0.000,B 0.000,C 90.000,E1 23.590} C_DIS
LIN {X -0.038,Y -539.430,Z 1410.927,A 0.000,B 0.000,C 90.000,E1 22.898} C_DIS
LIN {X -0.225,Y -533.367,Z 1410.923,A 0.000,B 0.000,C 90.000,E1 22.206} C_DIS
LIN {X -0.102,Y -525.739,Z 1410.918,A 0.000,B 0.000,C 90.000,E1 21.334} C_DIS
LIN {X -0.270,Y -515.535,Z 1410.912,A 0.000,B 0.000,C 90.000,E1 20.248} C_DIS
LIN {X 0.150,Y -504.696,Z 1410.906,A 0.000,B 0.000,C 90.000,E1 19.087} C_DIS
LIN {X -0.030,Y -492.565,Z 1410.899,A 0.000,B 0.000,C 90.000,E1 17.873} C_DIS
LIN {X -0.147,Y -477.438,Z 1410.891,A 0.000,B 0.000,C 90.000,E1 16.315} C_DIS
LIN {X 0.141,Y -465.117,Z 1410.883,A 0.000,B 0.000,C 90.000,E1 14.954} C_DIS
LIN {X 0.143,Y -452.767,Z 1410.876,A 0.000,B 0.000,C 90.000,E1 13.592} C_DIS
LIN {X 0.026,Y -434.855,Z 1410.865,A 0.000,B 0.000,C 90.000,E1 11.591} C_DIS
LIN {X -0.049,Y -423.996,Z 1410.857,A 0.000,B 0.000,C 90.000,E1 10.310} C_DIS
LIN {X 0.027,Y -404.251,Z 1410.843,A 0.000,B 0.000,C 90.000,E1 7.757} C_DIS
LIN {X -0.058,Y -393.672,Z 1410.835,A 0.000,B 0.000,C 90.000,E1 6.372} C_DIS
LIN {X 0.138,Y -389.200,Z 1410.832,A 0.000,B 0.000,C 90.000,E1 5.682} C_DIS
LIN {X -0.017,Y -386.724,Z 1410.829,A 0.000,B 0.000,C 90.000,E1 5.220} C_DIS
LIN {X -0.055,Y -386.706,Z 1410.829,A 0.000,B 0.000,C 90.000,E1 5.220} C_DIS
LIN {X -0.105,Y -386.473,Z 1410.828,A 0.000,B 0.000,C 90.000,E1 5.049} C_DIS
LIN {X -0.143,Y -386.502,Z 1410.828,A 0.000,B 0.000,C 90.000,E1 5.049} C_DIS
LIN {X -0.075,Y -387.665,Z 1410.827,A 0.000,B 0.000,C 90.000,E1 4.821} C_DIS
LIN {X -0.130,Y -391.885,Z 1410.824,A 0.000,B 0.000,C 90.000,E1 4.302} C_DIS
LIN {X -0.040,Y -398.687,Z 1410.820,A 0.000,B 0.000,C 90.000,E1 3.555} C_DIS
LIN {X 0.179,Y -404.251,Z 1410.816,A 0.000,B 0.000,C 90.000,E1 2.865} C_DIS
LIN {X 0.201,Y -407.402,Z 1410.813,A 0.000,B 0.000,C 90.000,E1 2.350} C_DIS
LIN {X 0.171,Y -410.165,Z 1410.810,A 0.000,B 0.000,C 90.000,E1 1.835} C_DIS
LIN {X 0.173,Y -411.627,Z 1410.808,A 0.000,B 0.000,C 90.000,E1 1.489} C_DIS
LIN {X 0.170,Y -412.645,Z 1410.807,A 0.000,B 0.000,C 90.000,E1 1.146} C_DIS
LIN {X 0.168,Y -412.800,Z 1410.805,A 0.000,B 0.000,C 90.000,E1 0.802} C_DIS
LIN {X 0.053,Y -412.363,Z 1410.804,A 0.000,B 0.000,C 90.000,E1 0.688} C_DIS
LIN {X -0.091,Y -411.637,Z 1410.803,A 0.000,B 0.000,C 90.000,E1 0.630} C_DIS
LIN {X 0.062,Y -410.640,Z 1410.803,A 0.000,B 0.000,C 90.000,E1 0.573} C_DIS
LIN {X 0.031,Y -360.918,Z 1410.803,A 0.000,B 0.000,C 90.000,E1 0.573} C_DIS
LIN {X 0.000,Y -360.799,Z 1410.800,A 0.000,B 0.000,C 90.000,E1 360.000} C_DIS
LIN {X -0.053,Y -359.426,Z 1410.770,A 0.000,B 0.000,C 90.000,E1 354.546} C_DIS
LIN {X 0.070,Y -358.890,Z 1410.759,A 0.000,B 0.000,C 90.000,E1 352.648} C_DIS
LIN {X -0.020,Y -359.563,Z 1410.726,A 0.000,B 0.000,C 90.000,E1 346.645} C_DIS
LIN {X 0.001,Y -361.801,Z 1410.684,A 0.000,B 0.000,C 90.000,E1 339.135} C_DIS
LIN {X -0.154,Y -362.053,Z 1410.680,A 0.000,B 0.000,C 90.000,E1 338.411} C_DIS
LIN {X 0.189,Y -365.980,Z 1410.643,A 0.000,B 0.000,C 90.000,E1 331.641} C_DIS
LIN {X 0.029,Y -366.387,Z 1410.639,A 0.000,B 0.000,C 90.000,E1 330.923} C_DIS
LIN {X -0.031,Y -371.355,Z 1410.604,A 0.000,B 0.000,C 90.000,E1 324.642} C_DIS
LIN {X -0.043,Y -371.766,Z 1410.602,A 0.000,B 0.000,C 90.000,E1 324.276} C_DIS
LIN {X 0.013,Y -377.358,Z 1410.567,A 0.000,B 0.000,C 90.000,E1 318.038} C_DIS
LIN {X 0.012,Y -378.235,Z 1410.563,A 0.000,B 0.000,C 90.000,E1 317.310} C_DIS
LIN {X 0.002,Y -383.940,Z 1410.531,A 0.000,B 0.000,C 90.000,E1 311.515} C_DIS
LIN {X 0.088,Y -384.893,Z 1410.527,A 0.000,B 0.000,C 90.000,E1 310.782} C_DIS
LIN {X 0.262,Y -390.610,Z 1410.495,A 0.000,B 0.000,C 90.000,E1 305.025} C_DIS
LIN {X 0.106,Y -391.104,Z 1410.493,A 0.000,B 0.000,C 90.000,E1 304.692} C_DIS
LIN {X 0.022,Y -391.648,Z 1410.489,A 0.000,B 0.000,C 90.000,E1 303.992} C_DIS
LIN {X -0.080,Y -396.825,Z 1410.459,A 0.000,B 0.000,C 90.000,E1 298.693} C_DIS
LIN {X -0.210,Y -397.120,Z 1410.457,A 0.000,B 0.000,C 90.000,E1 298.359} C_DIS
LIN {X -0.055,Y -401.597,Z 1410.426,A 0.000,B 0.000,C 90.000,E1 292.717} C_DIS
LIN {X 0.222,Y -404.659,Z 1410.395,A 0.000,B 0.000,C 90.000,E1 287.094} C_DIS
LIN {X -0.079,Y -404.735,Z 1410.391,A 0.000,B 0.000,C 90.000,E1 286.441} C_DIS
LIN {X 0.214,Y -406.099,Z 1410.364,A 0.000,B 0.000,C 90.000,E1 281.535} C_DIS
LIN {X -0.176,Y -406.094,Z 1410.362,A 0.000,B 0.000,C 90.000,E1 281.243} C_DIS
LIN {X -0.097,Y -405.680,Z 1410.333,A 0.000,B 0.000,C 90.000,E1 276.024} C_DIS
LIN {X -0.165,Y -405.058,Z 1410.328,A 0.000,B 0.000,C 90.000,E1 274.992} C_DIS
LIN {X -0.060,Y -403.497,Z 1410.304,A 0.000,B 0.000,C 90.000,E1 270.802} C_DIS
LIN {X -0.092,Y -403.288,Z 1410.302,A 0.000,B 0.000,C 90.000,E1 270.458} C_DIS
LIN {X 0.091,Y -398.931,Z 1410.271,A 0.000,B 0.000,C 90.000,E1 264.837} C_DIS
LIN {X -0.040,Y -393.108,Z 1410.242,A 0.000,B 0.000,C 90.000,E1 259.567} C_DIS
LIN {X -0.079,Y -392.835,Z 1410.240,A 0.000,B 0.000,C 90.000,E1 259.218} C_DIS
LIN {X 0.034,Y -385.993,Z 1410.212,A 0.000,B 0.000,C 90.000,E1 254.212} C_DIS
LIN {X -0.026,Y -385.267,Z 1410.208,A 0.000,B 0.000,C 90.000,E1 253.504} C_DIS
LIN {X -0.004,Y -384.768,Z 1410.206,A 0.000,B 0.000,C 90.000,E1 253.142} C_DIS
LIN {X 0.221,Y -377.973,Z 1410.182,A 0.000,B 0.000,C 90.000,E1 248.773} C_DIS
LIN {X -0.044,Y -376.233,Z 1410.174,A 0.000,B 0.000,C 90.000,E1 247.358} C_DIS
LIN {X 0.057,Y -374.944,Z 1410.170,A 0.000,B 0.000,C 90.000,E1 246.613} C_DIS
LIN {X -0.208,Y -368.417,Z 1410.148,A 0.000,B 0.000,C 90.000,E1 242.615} C_DIS
LIN {X 0.097,Y -366.047,Z 1410.137,A 0.000,B 0.000,C 90.000,E1 240.717} C_DIS
LIN {X 0.004,Y -359.196,Z 1410.115,A 0.000,B 0.000,C 90.000,E1 236.628} C_DIS
LIN {X 0.021,Y -355.842,Z 1410.100,A 0.000,B 0.000,C 90.000,E1 233.989} C_DIS
LIN {X -0.173,Y -348.793,Z 1410.075,A 0.000,B 0.000,C 90.000,E1 229.461} C_DIS
LIN {X -0.097,Y -346.185,Z 1410.062,A 0.000,B 0.000,C 90.000,E1 227.148} C_DIS
LIN {X -0.088,Y -345.065,Z 1410.058,A 0.000,B 0.000,C 90.000,E1 226.377} C_DIS
LIN {X 0.094,Y -338.586,Z 1410.030,A 0.000,B 0.000,C 90.000,E1 221.310} C_DIS
LIN {X 0.094,Y -336.840,Z 1410.019,A 0.000,B 0.000,C 90.000,E1 219.358} C_DIS
LIN {X 0.014,Y -330.861,Z 1409.988,A 0.000,B 0.000,C 90.000,E1 213.865} C_DIS
LIN {X 0.149,Y -329.296,Z 1409.975,A 0.000,B 0.000,C 90.000,E1 211.465} C_DIS
LIN {X -0.154,Y -324.669,Z 1409.942,A 0.000,B 0.000,C 90.000,E1 205.540} C_DIS
LIN {X 0.174,Y -323.837,Z 1409.928,A 0.000,B 0.000,C 90.000,E1 203.078} C_DIS
LIN {X -0.017,Y -321.124,Z 1409.881,A 0.000,B 0.000,C 90.000,E1 194.662} C_DIS
LIN {X 0.138,Y -320.932,Z 1409.877,A 0.000,B 0.000,C 90.000,E1 193.828} C_DIS
LIN {X -0.076,Y -321.562,Z 1409.832,A 0.000,B 0.000,C 90.000,E1 185.796} C_DIS
LIN {X -0.111,Y -323.256,Z 1409.799,A 0.000,B 0.000,C 90.000,E1 179.885} C_DIS
LIN {X -0.172,Y -385.981,Z 1409.799,A 0.000,B 0.000,C 90.000,E1 179.885} C_DIS
LIN {X 0.138,Y -386.512,Z 1409.799,A 0.000,B 0.000,C 90.000,E1 179.828} C_DIS
LIN {X -0.171,Y -387.794,Z 1409.799,A 0.000,B 0.000,C 90.000,E1 179.771} C_DIS
LIN {X 0.005,Y -388.350,Z 1409.797,A 0.000,B 0.000,C 90.000,E1 179.484} C_DIS
LIN {X -0.089,Y -387.849,Z 1409.795,A 0.000,B 0.000,C 90.000,E1 179.141} C_DIS
LIN {X -0.181,Y -386.782,Z 1409.793,A 0.000,B 0.000,C 90.000,E1 178.797} C_DIS
LIN {X 0.110,Y -385.386,Z 1409.791,A 0.000,B 0.000,C 90.000,E1 178.396} C_DIS
LIN {X 0.180,Y -380.187,Z 1409.785,A 0.000,B 0.000,C 90.000,E1 177.306} C_DIS
LIN {X -0.189,Y -374.246,Z 1409.779,A 0.000,B 0.000,C 90.000,E1 176.274} C_DIS
LIN {X 0.058,Y -367.295,Z 1409.772,A 0.000,B 0.000,C 90.000,E1 174.951} C_DIS
LIN {X -0.069,Y -358.302,Z 1409.762,A 0.000,B 0.000,C 90.000,E1 173.109} C_DIS
LIN {X -0.180,Y -354.078,Z 1409.756,A 0.000,B 0.000,C 90.000,E1 172.186} C_DIS
LIN {X 0.138,Y -351.291,Z 1409.752,A 0.000,B 0.000,C 90.000,E1 171.376} C_DIS
LIN {X -0.060,Y -350.055,Z 1409.750,A 0.000,B 0.000,C 90.000,E1 171.027} C_DIS
LIN {X 0.084,Y -349.152,Z 1409.748,A 0.000,B 0.000,C 90.000,E1 170.622} C_DIS
LIN {X 0.011,Y -348.985,Z 1409.747,A 0.000,B 0.000,C 90.000,E1 170.443} C_DIS
LIN {X 0.026,Y -349.066,Z 1409.745,A 0.000,B 0.000,C 90.000,E1 170.151} C_DIS
LIN {X 0.007,Y -349.077,Z 1409.745,A 0.000,B 0.000,C 90.000,E1 170.151} C_DIS
LIN {X 0.045,Y -351.443,Z 1409.742,A 0.000,B 0.000,C 90.000,E1 169.577} C_DIS
LIN {X -0.183,Y -357.121,Z 1409.737,A 0.000,B 0.000,C 90.000,E1 168.757} C_DIS
LIN {X -0.125,Y -362.731,Z 1409.733,A 0.000,B 0.000,C 90.000,E1 167.993} C_DIS
LIN {X 0.069,Y -374.304,Z 1409.725,A 0.000,B 0.000,C 90.000,E1 166.533} C_DIS
LIN {X 0.210,Y -387.518,Z 1409.717,A 0.000,B 0.000,C 90.000,E1 165.046} C_DIS
LIN {X 0.124,Y -399.541,Z 1409.711,A 0.000,B 0.000,C 90.000,E1 163.866} C_DIS
LIN {X -0.004,Y -416.771,Z 1409.702,A 0.000,B 0.000,C 90.000,E1 162.362} C_DIS
LIN {X 0.056,Y -427.701,Z 1409.697,A 0.000,B 0.000,C 90.000,E1 161.456} C_DIS
LIN {X 0.162,Y -440.309,Z 1409.691,A 0.000,B 0.000,C 90.000,E1 160.423} C_DIS
LIN {X -0.109,Y -451.128,Z 1409.687,A 0.000,B 0.000,C 90.000,E1 159.571} C_DIS
LIN {X -0.214,Y -461.440,Z 1409.682,A 0.000,B 0.000,C 90.000,E1 158.720} C_DIS
LIN {X 0.141,Y -470.374,Z 1409.677,A 0.000,B 0.000,C 90.000,E1 157.922} C_DIS
LIN {X -0.176,Y -482.028,Z 1409.672,A 0.000,B 0.000,C 90.000,E1 156.922} C_DIS
LIN {X 0.107,Y -489.181,Z 1409.668,A 0.000,B 0.000,C 90.000,E1 156.230} C_DIS
LIN {X 0.174,Y -497.670,Z 1409.664,A 0.000,B 0.000,C 90.000,E1 155.409} C_DIS
LIN {X 0.159,Y -504.359,Z 1409.660,A 0.000,B 0.000,C 90.000,E1 154.717} C_DIS
LIN {X 0.103,Y -509.582,Z 1409.656,A 0.000,B 0.000,C 90.000,E1 154.152} C_DIS
LIN {X 0.096,Y -513.432,Z 1409.654,A 0.000,B 0.000,C 90.000,E1 153.717} C_DIS
LIN {X -0.060,Y -519.343,Z 1409.650,A 0.000,B 0.000,C 90.000,E1 152.999} C_DIS
LIN {X 0.143,Y -522.702,Z 1409.648,A 0.000,B 0.000,C 90.000,E1 152.538} C_DIS
LIN {X -0.033,Y -526.782,Z 1409.644,A 0.000,B 0.000,C 90.000,E1 151.975} C_DIS
LIN {X 0.065,Y -530.390,Z 1409.641,A 0.000,B 0.000,C 90.000,E1 151.385} C_DIS
LIN {X 0.191,Y -533.607,Z 1409.638,A 0.000,B 0.000,C 90.000,E1 150.795} C_DIS
LIN {X 0.200,Y -536.994,Z 1409.634,A 0.000,B 0.000,C 90.000,E1 150.078} C_DIS
LIN {X -0.230,Y -539.923,Z 1409.630,A 0.000,B 0.000,C 90.000,E1 149.410} C_DIS
LIN {X -0.041,Y -542.000,Z 1409.627,A 0.000,B 0.000,C 90.000,E1 148.820} C_DIS
LIN {X -0.015,Y -543.897,Z 1409.624,A 0.000,B 0.000,C 90.000,E1 148.250} C_DIS
LIN {X 0.232,Y -546.382,Z 1409.619,A 0.000,B 0.000,C 90.000,E1 147.375} C_DIS
LIN {X 0.006,Y -547.877,Z 1409.616,A 0.000,B 0.000,C 90.000,E1 146.834} C_DIS
LIN {X -0.165,Y -549.784,Z 1409.611,A 0.000,B 0.000,C 90.000,E1 146.008} C_DIS
LIN {X -0.318,Y -551.415,Z 1409.606,A 0.000,B 0.000,C 90.000,E1 145.182} C_DIS
LIN {X -0.200,Y -552.354,Z 1409.603,A 0.000,B 0.000,C 90.000,E1 144.609} C_DIS
LIN {X -0.003,Y -553.447,Z 1409.599,A 0.000,B 0.000,C 90.000,E1 143.749} C_DIS
LIN {X -0.126,Y -554.365,Z 1409.594,A 0.000,B 0.000,C 90.000,E1 142.924} C_DIS
LIN {X -0.202,Y -555.637,Z 1409.586,A 0.000,B 0.000,C 90.000,E1 141.537} C_DIS
LIN {X 0.100,Y -556.898,Z 1409.578,A 0.000,B 0.000,C 90.000,E1 140.114} C_DIS
LIN {X 0.059,Y -557.898,Z 1409.571,A 0.000,B 0.000,C 90.000,E1 138.728} C_DIS
LIN {X 0.346,Y -558.616,Z 1409.563,A 0.000,B 0.000,C 90.000,E1 137.310} C_DIS
LIN {X 0.200,Y -559.191,Z 1409.557,A 0.000,B 0.000,C 90.000,E1 136.215} C_DIS
LIN {X 0.116,Y -559.654,Z 1409.549,A 0.000,B 0.000,C 90.000,E1 134.838} C_DIS
LIN {X 0.039,Y -560.080,Z 1409.542,A 0.000,B 0.000,C 90.000,E1 133.461} C_DIS
LIN {X 0.242,Y -560.281,Z 1409.537,A 0.000,B 0.000,C 90.000,E1 132.609} C_DIS
LIN {X 0.041,Y -560.432,Z 1409.525,A 0.000,B 0.000,C 90.000,E1 130.415} C_DIS
LIN {X 0.277,Y -560.752,Z 1409.512,A 0.000,B 0.000,C 90.000,E1 128.177} C_DIS
LIN {X 0.215,Y -560.863,Z 1409.506,A 0.000,B 0.000,C 90.000,E1 127.076} C_DIS
LIN {X 0.004,Y -560.849,Z 1409.497,A 0.000,B 0.000,C 90.000,E1 125.438} C_DIS
LIN {X 0.151,Y -560.860,Z 1409.489,A 0.000,B 0.000,C 90.000,E1 124.040} C_DIS
LIN {X -0.056,Y -561.103,Z 1409.477,A 0.000,B 0.000,C 90.000,E1 121.848} C_DIS
LIN {X 0.296,Y -561.412,Z 1409.474,A 0.000,B 0.000,C 90.000,E1 121.258} C_DIS
LIN {X -0.031,Y -562.367,Z 1409.469,A 0.000,B 0.000,C 90.000,E1 120.463} C_DIS
LIN {X -0.014,Y -562.931,Z 1409.467,A 0.000,B 0.000,C 90.000,E1 120.129} C_DIS
LIN {X -0.056,Y -562.940,Z 1409.467,A 0.000,B 0.000,C 90.000,E1 120.129} C_DIS
LIN {X 0.026,Y -564.647,Z 1409.466,A 0.000,B 0.000,C 90.000,E1 119.873} C_DIS
LIN {X -0.104,Y -568.882,Z 1409.465,A 0.000,B 0.000,C 90.000,E1 119.716} C_DIS
LIN {X 0.146,Y -571.820,Z 1409.465,A 0.000,B 0.000,C 90.000,E1 119.617} C_DIS
LIN {X -0.024,Y -574.923,Z 1409.464,A 0.000,B 0.000,C 90.000,E1 119.589} C_DIS
LIN {X -0.010,Y -579.820,Z 1409.464,A 0.000,B 0.000,C 90.000,E1 119.461} C_DIS
LIN {X 0.277,Y -582.644,Z 1409.463,A 0.000,B 0.000,C 90.000,E1 119.333} C_DIS
LIN {X 0.332,Y -585.175,Z 1409.463,A 0.000,B 0.000,C 90.000,E1 119.205} C_DIS
LIN {X 0.007,Y -588.150,Z 1409.462,A 0.000,B 0.000,C 90.000,E1 119.077} C_DIS
LIN {X -0.231,Y -592.074,Z 1409.460,A 0.000,B 0.000,C 90.000,E1 118.821} C_DIS
LIN {X 0.150,Y -594.640,Z 1409.459,A 0.000,B 0.000,C 90.000,E1 118.565} C_DIS
LIN {X -0.150,Y -597.238,Z 1409.458,A 0.000,B 0.000,C 90.000,E1 118.359} C_DIS
LIN {X -0.076,Y -602.169,Z 1409.455,A 0.000,B 0.000,C 90.000,E1 117.847} C_DIS
LIN {X -0.176,Y -606.156,Z 1409.452,A 0.000,B 0.000,C 90.000,E1 117.334} C_DIS
LIN {X -0.031,Y -609.717,Z 1409.448,A 0.000,B 0.000,C 90.000,E1 116.668} C_DIS
LIN {X -0.074,Y -610.362,Z 1409.447,A 0.000,B 0.000,C 90.000,E1 116.411} C_DIS
LIN {X -0.155,Y -611.174,Z 1409.444,A 0.000,B 0.000,C 90.000,E1 115.899} C_DIS
LIN {X 0.321,Y -610.809,Z 1409.441,A 0.000,B 0.000,C 90.000,E1 115.335} C_DIS
LIN {X 0.283,Y -610.140,Z 1409.440,A 0.000,B 0.000,C 90.000,E1 115.079} C_DIS
LIN {X -0.053,Y -607.206,Z 1409.437,A 0.000,B 0.000,C 90.000,E1 114.591} C_DIS
LIN {X -0.100,Y -603.996,Z 1409.435,A 0.000,B 0.000,C 90.000,E1 114.335} C_DIS
LIN {X -0.165,Y -603.094,Z 1409.434,A 0.000,B 0.000,C 90.000,E1 114.207} C_DIS
LIN {X -0.196,Y -601.924,Z 1409.434,A 0.000,B 0.000,C 90.000,E1 114.079} C_DIS
LIN {X 0.113,Y -595.004,Z 1409.432,A 0.000,B 0.000,C 90.000,E1 113.643} C_DIS
LIN {X -0.083,Y -593.116,Z 1409.431,A 0.000,B 0.000,C 90.000,E1 113.567} C_DIS
LIN {X 0.281,Y -579.333,Z 1409.428,A 0.000,B 0.000,C 90.000,E1 112.950} C_DIS
LIN {X -0.336,Y -578.246,Z 1409.427,A 0.000,B 0.000,C 90.000,E1 112.898} C_DIS
LIN {X 0.157,Y -578.240,Z 1409.427,A 0.000,B 0.000,C 90.000,E1 112.845} C_DIS
LIN {X -0.158,Y -578.580,Z 1409.427,A 0.000,B 0.000,C 90.000,E1 112.823} C_DIS
LIN {X -0.195,Y -580.091,Z 1409.426,A 0.000,B 0.000,C 90.000,E1 112.695} C_DIS
LIN {X -0.158,Y -583.912,Z 1409.425,A 0.000,B 0.000,C 90.000,E1 112.461} C_DIS
LIN {X -0.334,Y -589.622,Z 1409.423,A 0.000,B 0.000,C 90.000,E1 112.153} C_DIS
LIN {X -0.060,Y -594.157,Z 1409.421,A 0.000,B 0.000,C 90.000,E1 111.844} C_DIS
LIN {X 0.297,Y -599.933,Z 1409.419,A 0.000,B 0.000,C 90.000,E1 111.408} C_DIS
LIN {X 0.266,Y -605.386,Z 1409.417,A 0.000,B 0.000,C 90.000,E1 110.972} C_DIS
LIN {X -0.120,Y -609.445,Z 1409.415,A 0.000,B 0.000,C 90.000,E1 110.663} C_DIS
LIN {X 0.006,Y -614.499,Z 1409.412,A 0.000,B 0.000,C 90.000,E1 110.174} C_DIS
LIN {X -0.084,Y -619.260,Z 1409.409,A 0.000,B 0.000,C 90.000,E1 109.685} C_DIS
LIN {X 0.375,Y -623.646,Z 1409.407,A 0.000,B 0.000,C 90.000,E1 109.141} C_DIS
LIN {X -0.077,Y -629.424,Z 1409.402,A 0.000,B 0.000,C 90.000,E1 108.417} C_DIS
LIN {X 0.124,Y -633.565,Z 1409.399,A 0.000,B 0.000,C 90.000,E1 107.764} C_DIS
LIN {X -0.055,Y -637.006,Z 1409.395,A 0.000,B 0.000,C 90.000,E1 107.149} C_DIS
LIN {X -0.233,Y -638.205,Z 1409.394,A 0.000,B 0.000,C 90.000,E1 106.913} C_DIS
LIN {X 0.051,Y -640.937,Z 1409.390,A 0.000,B 0.000,C 90.000,E1 106.134} C_DIS
LIN {X -0.273,Y -642.097,Z 1409.387,A 0.000,B 0.000,C 90.000,E1 105.662} C_DIS
LIN {X -0.108,Y -643.662,Z 1409.381,A 0.000,B 0.000,C 90.000,E1 104.647} C_DIS
LIN {X -0.086,Y -644.892,Z 1409.376,A 0.000,B 0.000,C 90.000,E1 103.647} C_DIS
LIN {X 0.246,Y -645.358,Z 1409.373,A 0.000,B 0.000,C 90.000,E1 103.119} C_DIS
LIN {X -0.193,Y -645.540,Z 1409.369,A 0.000,B 0.000,C 90.000,E1 102.411} C_DIS
LIN {X 0.291,Y -645.559,Z 1409.368,A 0.000,B 0.000,C 90.000,E1 102.119} C_DIS
LIN {X -0.280,Y -645.063,Z 1409.363,A 0.000,B 0.000,C 90.000,E1 101.422} C_DIS
LIN {X 0.056,Y -644.527,Z 1409.361,A 0.000,B 0.000,C 90.000,E1 100.894} C_DIS
LIN {X 0.116,Y -643.248,Z 1409.356,A 0.000,B 0.000,C 90.000,E1 100.141} C_DIS
LIN {X -0.198,Y -642.151,Z 1409.354,A 0.000,B 0.000,C 90.000,E1 99.670} C_DIS
LIN {X 0.006,Y -640.795,Z 1409.351,A 0.000,B 0.000,C 90.000,E1 99.151} C_DIS
LIN {X 0.301,Y -639.240,Z 1409.348,A 0.000,B 0.000,C 90.000,E1 98.624} C_DIS
LIN {X -0.143,Y -637.436,Z 1409.345,A 0.000,B 0.000,C 90.000,E1 98.163} C_DIS
LIN {X -0.155,Y -634.181,Z 1409.341,A 0.000,B 0.000,C 90.000,E1 97.409} C_DIS
LIN {X -0.137,Y -631.143,Z 1409.338,A 0.000,B 0.000,C 90.000,E1 96.777} C_DIS
LIN {X -0.143,Y -627.770,Z 1409.334,A 0.000,B 0.000,C 90.000,E1 96.144} C_DIS
LIN {X -0.178,Y -624.107,Z 1409.331,A 0.000,B 0.000,C 90.000,E1 95.511} C_DIS
LIN {X -0.092,Y -620.830,Z 1409.328,A 0.000,B 0.000,C 90.000,E1 94.992} C_DIS
LIN {X 0.276,Y -619.112,Z 1409.326,A 0.000,B 0.000,C 90.000,E1 94.702} C_DIS
LIN {X 0.274,Y -615.006,Z 1409.323,A 0.000,B 0.000,C 90.000,E1 94.188} C_DIS
LIN {X -0.157,Y -611.336,Z 1409.321,A 0.000,B 0.000,C 90.000,E1 93.841} C_DIS
LIN {X 0.160,Y -608.728,Z 1409.320,A 0.000,B 0.000,C 90.000,E1 93.555} C_DIS
LIN {X -0.162,Y -601.861,Z 1409.317,A 0.000,B 0.000,C 90.000,E1 92.980} C_DIS
LIN {X -0.093,Y -595.121,Z 1409.313,A 0.000,B 0.000,C 90.000,E1 92.407} C_DIS
LIN {X -0.045,Y -590.799,Z 1409.312,A 0.000,B 0.000,C 90.000,E1 92.064} C_DIS
LIN {X -0.149,Y -584.324,Z 1409.309,A 0.000,B 0.000,C 90.000,E1 91.661} C_DIS
LIN {X 0.202,Y -577.761,Z 1409.307,A 0.000,B 0.000,C 90.000,E1 91.260} C_DIS
LIN {X -0.117,Y -576.570,Z 1409.307,A 0.000,B 0.000,C 90.000,E1 91.203} C_DIS
LIN {X 0.147,Y -573.816,Z 1409.305,A 0.000,B 0.000,C 90.000,E1 90.917} C_DIS
LIN {X 0.107,Y -573.795,Z 1409.305,A 0.000,B 0.000,C 90.000,E1 90.917} C_DIS
LIN {X 0.257,Y -573.162,Z 1409.304,A 0.000,B 0.000,C 90.000,E1 90.688} C_DIS
LIN {X 0.042,Y -573.000,Z 1409.303,A 0.000,B 0.000,C 90.000,E1 90.573} C_DIS
LIN {X -0.247,Y -572.994,Z 1409.300,A 0.000,B 0.000,C 90.000,E1 90.057} C_DIS
LIN {X 0.195,Y -574.639,Z 1409.290,A 0.000,B 0.000,C 90.000,E1 88.108} C_DIS
LIN {X -0.045,Y -576.114,Z 1409.281,A 0.000,B 0.000,C 90.000,E1 86.502} C_DIS
LIN {X 0.118,Y -578.229,Z 1409.269,A 0.000,B 0.000,C 90.000,E1 84.318} C_DIS
LIN {X 0.251,Y -580.345,Z 1409.258,A 0.000,B 0.000,C 90.000,E1 82.413} C_DIS
LIN {X 0.284,Y -582.231,Z 1409.249,A 0.000,B 0.000,C 90.000,E1 80.792} C_DIS
LIN {X -0.124,Y -584.051,Z 1409.240,A 0.000,B 0.000,C 90.000,E1 79.218} C_DIS
LIN {X -0.174,Y -585.400,Z 1409.233,A 0.000,B 0.000,C 90.000,E1 77.881} C_DIS
LIN {X 0.295,Y -586.697,Z 1409.224,A 0.000,B 0.000,C 90.000,E1 76.228} C_DIS
LIN {X -0.098,Y -587.373,Z 1409.219,A 0.000,B 0.000,C 90.000,E1 75.463} C_DIS
LIN {X 0.159,Y -588.234,Z 1409.212,A 0.000,B 0.000,C 90.000,E1 74.102} C_DIS
LIN {X -0.289,Y -589.112,Z 1409.203,A 0.000,B 0.000,C 90.000,E1 72.543} C_DIS
LIN {X -0.082,Y -589.744,Z 1409.197,A 0.000,B 0.000,C 90.000,E1 71.456} C_DIS
LIN {X -0.206,Y -590.886,Z 1409.185,A 0.000,B 0.000,C 90.000,E1 69.337} C_DIS
LIN {X -0.328,Y -592.018,Z 1409.175,A 0.000,B 0.000,C 90.000,E1 67.486} C_DIS
LIN {X -0.094,Y -593.128,Z 1409.166,A 0.000,B 0.000,C 90.000,E1 65.869} C_DIS
LIN {X -0.225,Y -594.538,Z 1409.156,A 0.000,B 0.000,C 90.000,E1 64.024} C_DIS
LIN {X 0.127,Y -595.605,Z 1409.148,A 0.000,B 0.000,C 90.000,E1 62.666} C_DIS
LIN {X -0.106,Y -596.873,Z 1409.139,A 0.000,B 0.000,C 90.000,E1 61.101} C_DIS
LIN {X -0.235,Y -598.074,Z 1409.132,A 0.000,B 0.000,C 90.000,E1 59.793} C_DIS
LIN {X -0.132,Y -599.550,Z 1409.123,A 0.000,B 0.000,C 90.000,E1 58.201} C_DIS
LIN {X -0.194,Y -600.964,Z 1409.115,A 0.000,B 0.000,C 90.000,E1 56.628} C_DIS
LIN {X 0.019,Y -602.659,Z 1409.104,A 0.000,B 0.000,C 90.000,E1 54.769} C_DIS
LIN {X -0.137,Y -604.020,Z 1409.096,A 0.000,B 0.000,C 90.000,E1 53.210} C_DIS
LIN {X -0.164,Y -604.967,Z 1409.088,A 0.000,B 0.000,C 90.000,E1 51.904} C_DIS
LIN {X -0.057,Y -605.681,Z 1409.083,A 0.000,B 0.000,C 90.000,E1 50.848} C_DIS
LIN {X -0.059,Y -606.379,Z 1409.075,A 0.000,B 0.000,C 90.000,E1 49.542} C_DIS
LIN {X 0.066,Y -606.709,Z 1409.069,A 0.000,B 0.000,C 90.000,E1 48.485} C_DIS
LIN {X -0.002,Y -606.847,Z 1409.062,A 0.000,B 0.000,C 90.000,E1 47.187} C_DIS
LIN {X -0.098,Y -606.989,Z 1409.055,A 0.000,B 0.000,C 90.000,E1 45.891} C_DIS
LIN {X 0.007,Y -606.870,Z 1409.049,A 0.000,B 0.000,C 90.000,E1 44.838} C_DIS
LIN {X -0.082,Y -606.486,Z 1409.042,A 0.000,B 0.000,C 90.000,E1 43.542} C_DIS
LIN {X 0.039,Y -605.967,Z 1409.036,A 0.000,B 0.000,C 90.000,E1 42.486} C_DIS
LIN {X 0.369,Y -605.179,Z 1409.029,A 0.000,B 0.000,C 90.000,E1 41.148} C_DIS
LIN {X -0.322,Y -603.797,Z 1409.020,A 0.000,B 0.000,C 90.000,E1 39.644} C_DIS
LIN {X 0.016,Y -602.386,Z 1409.013,A 0.000,B 0.000,C 90.000,E1 38.302} C_DIS
LIN {X -0.051,Y -600.612,Z 1409.006,A 0.000,B 0.000,C 90.000,E1 36.996} C_DIS
LIN {X 0.087,Y -598.886,Z 1409.000,A 0.000,B 0.000,C 90.000,E1 35.931} C_DIS
LIN {X -0.143,Y -596.885,Z 1408.994,A 0.000,B 0.000,C 90.000,E1 34.898} C_DIS
LIN {X 0.318,Y -595.799,Z 1408.991,A 0.000,B 0.000,C 90.000,E1 34.326} C_DIS
LIN {X -0.061,Y -592.610,Z 1408.984,A 0.000,B 0.000,C 90.000,E1 33.038} C_DIS
LIN {X 0.244,Y -590.451,Z 1408.979,A 0.000,B 0.000,C 90.000,E1 32.212} C_DIS
LIN {X -0.291,Y -588.044,Z 1408.975,A 0.000,B 0.000,C 90.000,E1 31.465} C_DIS
LIN {X -0.346,Y -585.342,Z 1408.970,A 0.000,B 0.000,C 90.000,E1 30.669} C_DIS
LIN {X -0.298,Y -583.261,Z 1408.967,A 0.000,B 0.000,C 90.000,E1 30.129} C_DIS
LIN {X 0.102,Y -579.756,Z 1408.963,A 0.000,B 0.000,C 90.000,E1 29.283} C_DIS
LIN {X 0.032,Y -576.612,Z 1408.959,A 0.000,B 0.000,C 90.000,E1 28.615} C_DIS
LIN {X -0.345,Y -573.097,Z 1408.955,A 0.000,B 0.000,C 90.000,E1 27.975} C_DIS
LIN {X -0.061,Y -568.714,Z 1408.951,A 0.000,B 0.000,C 90.000,E1 27.129} C_DIS
LIN {X 0.073,Y -563.135,Z 1408.945,A 0.000,B 0.000,C 90.000,E1 26.155} C_DIS
LIN {X -0.009,Y -557.862,Z 1408.941,A 0.000,B 0.000,C 90.000,E1 25.335} C_DIS
LIN {X -0.033,Y -553.124,Z 1408.937,A 0.000,B 0.000,C 90.000,E1 24.643} C_DIS
LIN {X 0.018,Y -549.097,Z 1408.934,A 0.000,B 0.000,C 90.000,E1 24.079} C_DIS
LIN {X -0.210,Y -542.540,Z 1408.929,A 0.000,B 0.000,C 90.000,E1 23.259} C_DIS
LIN {X 0.260,Y -537.890,Z 1408.926,A 0.000,B 0.000,C 90.000,E1 22.642} C_DIS
LIN {X -0.013,Y -531.833,Z 1408.922,A 0.000,B 0.000,C 90.000,E1 21.972} C_DIS
LIN {X -0.099,Y -525.621,Z 1408.918,A 0.000,B 0.000,C 90.000,E1 21.280} C_DIS
LIN {X -0.116,Y -515.360,Z 1408.912,A 0.000,B 0.000,C 90.000,E1 20.174} C_DIS
LIN {X -0.088,Y -504.797,Z 1408.906,A 0.000,B 0.000,C 90.000,E1 19.087} C_DIS
LIN {X -0.204,Y -494.022,Z 1408.900,A 0.000,B 0.000,C 90.000,E1 18.000} C_DIS
LIN {X 0.149,Y -477.611,Z 1408.891,A 0.000,B 0.000,C 90.000,E1 16.260} C_DIS
LIN {X -0.073,Y -464.029,Z 1408.882,A 0.000,B 0.000,C 90.000,E1 14.828} C_DIS
LIN {X -0.037,Y -451.676,Z 1408.875,A 0.000,B 0.000,C 90.000,E1 13.467} C_DIS
LIN {X 0.089,Y -435.093,Z 1408.865,A 0.000,B 0.000,C 90.000,E1 11.591} C_DIS
LIN {X 0.163,Y -416.387,Z 1408.852,A 0.000,B 0.000,C 90.000,E1 9.321} C_DIS
LIN {X -0.055,Y -403.267,Z 1408.843,A 0.000,B 0.000,C 90.000,E1 7.644} C_DIS
LIN {X -0.056,Y -392.796,Z 1408.835,A 0.000,B 0.000,C 90.000,E1 6.258} C_DIS
LIN {X -0.139,Y -389.268,Z 1408.832,A 0.000,B 0.000,C 90.000,E1 5.739} C_DIS
LIN {X -0.141,Y -387.045,Z 1408.829,A 0.000,B 0.000,C 90.000,E1 5.277} C_DIS
LIN {X -0.179,Y -387.040,Z 1408.829,A 0.000,B 0.000,C 90.000,E1 5.277} C_DIS
LIN {X -0.004,Y -386.986,Z 1408.828,A 0.000,B 0.000,C 90.000,E1 5.106} C_DIS
LIN {X -0.041,Y -387.010,Z 1408.828,A 0.000,B 0.000,C 90.000,E1 5.106} C_DIS
LIN {X 0.036,Y -388.518,Z 1408.827,A 0.000,B 0.000,C 90.000,E1 4.821} C_DIS
LIN {X 0.073,Y -392.426,Z 1408.824,A 0.000,B 0.000,C 90.000,E1 4.359} C_DIS
LIN {X 0.062,Y -398.749,Z 1408.821,A 0.000,B 0.000,C 90.000,E1 3.726} C_DIS
LIN {X 0.174,Y -404.521,Z 1408.817,A 0.000,B 0.000,C 90.000,E1 3.094} C_DIS
LIN {X -0.037,Y -408.106,Z 1408.815,A 0.000,B 0.000,C 90.000,E1 2.636} C_DIS
LIN {X -0.066,Y -411.568,Z 1408.812,A 0.000,B 0.000,C 90.000,E1 2.121} C_DIS
LIN {X -0.058,Y -414.593,Z 1408.809,A 0.000,B 0.000,C 90.000,E1 1.604} C_DIS
LIN {X -0.038,Y -417.685,Z 1408.805,A 0.000,B 0.000,C 90.000,E1 0.917} C_DIS
LIN {X -0.029,Y -418.346,Z 1408.804,A 0.000,B 0.000,C 90.000,E1 0.745} C_DIS
LIN {X -0.005,Y -419.389,Z 1408.802,A 0.000,B 0.000,C 90.000,E1 0.401} C_DIS
LIN {X 0.022,Y -419.894,Z 1408.800,A 0.000,B 0.000,C 90.000,E1 0.057} C_DIS
LIN {X 0.000,Y -419.884,Z 1408.800,A 0.000,B 0.000,C 90.000,E1 360.000} C_DIS
LIN {X 0.159,Y -419.291,Z 1408.799,A 0.000,B 0.000,C 90.000,E1 359.771} C_DIS
LIN {X -0.162,Y -418.911,Z 1408.799,A 0.000,B 0.000,C 90.000,E1 359.771} C_DIS
LIN {X -0.050,Y -418.217,Z 1408.798,A 0.000,B 0.000,C 90.000,E1 359.714} C_DIS
LIN {X -0.196,Y -415.510,Z 1408.798,A 0.000,B 0.000,C 90.000,E1 359.714} C_DIS
LIN {X 0.180,Y -408.796,Z 1408.798,A 0.000,B 0.000,C 90.000,E1 359.656} C_DIS
LIN {X 0.142,Y -402.298,Z 1408.798,A 0.000,B 0.000,C 90.000,E1 359.656} C_DIS
LIN {X 0.105,Y -395.999,Z 1408.798,A 0.000,B 0.000,C 90.000,E1 359.656} C_DIS
LIN {X 0.068,Y -389.892,Z 1408.798,A 0.000,B 0.000,C 90.000,E1 359.656} C_DIS
LIN {X 0.028,Y -383.090,Z 1408.798,A 0.000,B 0.000,C 90.000,E1 359.656} C_DIS
LIN {X -0.010,Y -376.516,Z 1408.798,A 0.000,B 0.000,C 90.000,E1 359.656} C_DIS
LIN {X -0.047,Y -370.159,Z 1408.798,A 0.000,B 0.000,C 90.000,E1 359.656} C_DIS
LIN {X -0.083,Y -364.009,Z 1408.798,A 0.000,B 0.000,C 90.000,E1 359.656} C_DIS
LIN {X -0.119,Y -360.603,Z 1408.798,A 0.000,B 0.000,C 90.000,E1 359.656} C_DIS
LIN {X 0.136,Y -359.424,Z 1408.770,A 0.000,B 0.000,C 90.000,E1 354.552} C_DIS
LIN {X 0.142,Y -359.229,Z 1408.766,A 0.000,B 0.000,C 90.000,E1 353.799} C_DIS
LIN {X -0.147,Y -359.547,Z 1408.726,A 0.000,B 0.000,C 90.000,E1 346.700} C_DIS
LIN {X 0.148,Y -361.980,Z 1408.682,A 0.000,B 0.000,C 90.000,E1 338.773} C_DIS
LIN {X -0.082,Y -365.945,Z 1408.643,A 0.000,B 0.000,C 90.000,E1 331.719} C_DIS
LIN {X 0.172,Y -366.226,Z 1408.641,A 0.000,B 0.000,C 90.000,E1 331.307} C_DIS
LIN {X -0.107,Y -371.315,Z 1408.604,A 0.000,B 0.000,C 90.000,E1 324.689} C_DIS
LIN {X -0.120,Y -371.739,Z 1408.602,A 0.000,B 0.000,C 90.000,E1 324.322} C_DIS
LIN {X -0.028,Y -377.786,Z 1408.565,A 0.000,B 0.000,C 90.000,E1 317.715} C_DIS
LIN {X 0.239,Y -378.213,Z 1408.563,A 0.000,B 0.000,C 90.000,E1 317.310} C_DIS
LIN {X -0.024,Y -383.894,Z 1408.531,A 0.000,B 0.000,C 90.000,E1 311.553} C_DIS
LIN {X 0.026,Y -384.865,Z 1408.527,A 0.000,B 0.000,C 90.000,E1 310.825} C_DIS
LIN {X -0.052,Y -390.565,Z 1408.495,A 0.000,B 0.000,C 90.000,E1 305.105} C_DIS
LIN {X 0.014,Y -391.057,Z 1408.493,A 0.000,B 0.000,C 90.000,E1 304.739} C_DIS
LIN {X -0.140,Y -391.409,Z 1408.491,A 0.000,B 0.000,C 90.000,E1 304.405} C_DIS
LIN {X 0.151,Y -396.781,Z 1408.460,A 0.000,B 0.000,C 90.000,E1 298.693} C_DIS
LIN {X 0.021,Y -397.105,Z 1408.458,A 0.000,B 0.000,C 90.000,E1 298.359} C_DIS
LIN {X -0.193,Y -401.567,Z 1408.426,A 0.000,B 0.000,C 90.000,E1 292.770} C_DIS
LIN {X -0.052,Y -404.629,Z 1408.395,A 0.000,B 0.000,C 90.000,E1 287.166} C_DIS
LIN {X 0.050,Y -404.755,Z 1408.393,A 0.000,B 0.000,C 90.000,E1 286.804} C_DIS
LIN {X 0.049,Y -406.081,Z 1408.365,A 0.000,B 0.000,C 90.000,E1 281.591} C_DIS
LIN {X 0.057,Y -406.108,Z 1408.363,A 0.000,B 0.000,C 90.000,E1 281.243} C_DIS
LIN {X 0.093,Y -405.672,Z 1408.334,A 0.000,B 0.000,C 90.000,E1 276.030} C_DIS
LIN {X 0.102,Y -405.306,Z 1408.330,A 0.000,B 0.000,C 90.000,E1 275.334} C_DIS
LIN {X 0.172,Y -403.517,Z 1408.305,A 0.000,B 0.000,C 90.000,E1 270.802} C_DIS
LIN {X 0.140,Y -403.308,Z 1408.303,A 0.000,B 0.000,C 90.000,E1 270.458} C_DIS
LIN {X -0.075,Y -398.962,Z 1408.272,A 0.000,B 0.000,C 90.000,E1 264.894} C_DIS
LIN {X 0.118,Y -393.134,Z 1408.242,A 0.000,B 0.000,C 90.000,E1 259.577} C_DIS
LIN {X 0.150,Y -392.868,Z 1408.240,A 0.000,B 0.000,C 90.000,E1 259.218} C_DIS
LIN {X -0.108,Y -386.029,Z 1408.213,A 0.000,B 0.000,C 90.000,E1 254.267} C_DIS
LIN {X -0.166,Y -385.300,Z 1408.209,A 0.000,B 0.000,C 90.000,E1 253.559} C_DIS
LIN {X -0.144,Y -384.830,Z 1408.207,A 0.000,B 0.000,C 90.000,E1 253.196} C_DIS
LIN {X -0.041,Y -378.017,Z 1408.182,A 0.000,B 0.000,C 90.000,E1 248.847} C_DIS
LIN {X 0.182,Y -376.271,Z 1408.174,A 0.000,B 0.000,C 90.000,E1 247.358} C_DIS
LIN {X -0.185,Y -375.707,Z 1408.172,A 0.000,B 0.000,C 90.000,E1 247.050} C_DIS
LIN {X -0.082,Y -368.976,Z 1408.150,A 0.000,B 0.000,C 90.000,E1 242.999} C_DIS
LIN {X -0.178,Y -366.113,Z 1408.138,A 0.000,B 0.000,C 90.000,E1 240.795} C_DIS
LIN {X 0.227,Y -359.246,Z 1408.115,A 0.000,B 0.000,C 90.000,E1 236.628} C_DIS
LIN {X -0.045,Y -355.905,Z 1408.100,A 0.000,B 0.000,C 90.000,E1 234.036} C_DIS
LIN {X 0.047,Y -348.840,Z 1408.075,A 0.000,B 0.000,C 90.000,E1 229.461} C_DIS
LIN {X 0.123,Y -346.221,Z 1408.062,A 0.000,B 0.000,C 90.000,E1 227.148} C_DIS
LIN {X 0.009,Y -345.743,Z 1408.060,A 0.000,B 0.000,C 90.000,E1 226.782} C_DIS
LIN {X -0.030,Y -339.022,Z 1408.032,A 0.000,B 0.000,C 90.000,E1 221.757} C_DIS
LIN {X 0.051,Y -336.878,Z 1408.019,A 0.000,B 0.000,C 90.000,E1 219.402} C_DIS
LIN {X -0.147,Y -331.212,Z 1407.991,A 0.000,B 0.000,C 90.000,E1 214.326} C_DIS
LIN {X -0.088,Y -329.316,Z 1407.975,A 0.000,B 0.000,C 90.000,E1 211.544} C_DIS
LIN {X -0.143,Y -324.884,Z 1407.944,A 0.000,B 0.000,C 90.000,E1 205.976} C_DIS
LIN {X -0.037,Y -323.847,Z 1407.929,A 0.000,B 0.000,C 90.000,E1 203.153} C_DIS
LIN {X -0.115,Y -321.119,Z 1407.882,A 0.000,B 0.000,C 90.000,E1 194.717} C_DIS
LIN {X 0.039,Y -320.945,Z 1407.877,A 0.000,B 0.000,C 90.000,E1 193.883} C_DIS
LIN {X 0.139,Y -321.544,Z 1407.832,A 0.000,B 0.000,C 90.000,E1 185.796} C_DIS
LIN {X -0.068,Y -322.679,Z 1407.805,A 0.000,B 0.000,C 90.000,E1 180.974} C_DIS
LIN {X -0.093,Y -324.048,Z 1407.805,A 0.000,B 0.000,C 90.000,E1 180.974} C_DIS
LIN {X -0.089,Y -392.917,Z 1407.804,A 0.000,B 0.000,C 90.000,E1 180.802} C_DIS
LIN {X 0.099,Y -394.881,Z 1407.803,A 0.000,B 0.000,C 90.000,E1 180.573} C_DIS
LIN {X -0.059,Y -395.049,Z 1407.802,A 0.000,B 0.000,C 90.000,E1 180.286} C_DIS
LIN {X -0.126,Y -394.424,Z 1407.800,A 0.000,B 0.000,C 90.000,E1 179.943} C_DIS
LIN {X -0.191,Y -393.389,Z 1407.798,A 0.000,B 0.000,C 90.000,E1 179.599} C_DIS
LIN {X 0.058,Y -390.581,Z 1407.794,A 0.000,B 0.000,C 90.000,E1 178.854} C_DIS
LIN {X -0.067,Y -388.361,Z 1407.791,A 0.000,B 0.000,C 90.000,E1 178.339} C_DIS
LIN {X 0.096,Y -384.069,Z 1407.786,A 0.000,B 0.000,C 90.000,E1 177.421} C_DIS
LIN {X -0.166,Y -379.258,Z 1407.781,A 0.000,B 0.000,C 90.000,E1 176.560} C_DIS
LIN {X -0.080,Y -369.148,Z 1407.771,A 0.000,B 0.000,C 90.000,E1 174.723} C_DIS
LIN {X 0.064,Y -358.333,Z 1407.758,A 0.000,B 0.000,C 90.000,E1 172.470} C_DIS
LIN {X -0.045,Y -354.321,Z 1407.753,A 0.000,B 0.000,C 90.000,E1 171.546} C_DIS
LIN {X -0.030,Y -350.970,Z 1407.747,A 0.000,B 0.000,C 90.000,E1 170.500} C_DIS
LIN {X 0.068,Y -350.612,Z 1407.745,A 0.000,B 0.000,C 90.000,E1 169.982} C_DIS
LIN {X 0.050,Y -350.611,Z 1407.744,A 0.000,B 0.000,C 90.000,E1 169.982} C_DIS
LIN {X -0.150,Y -351.603,Z 1407.743,A 0.000,B 0.000,C 90.000,E1 169.746} C_DIS
LIN {X 0.126,Y -352.177,Z 1407.742,A 0.000,B 0.000,C 90.000,E1 169.511} C_DIS
LIN {X 0.173,Y -356.562,Z 1407.738,A 0.000,B 0.000,C 90.000,E1 168.814} C_DIS
LIN {X -0.122,Y -362.036,Z 1407.734,A 0.000,B 0.000,C 90.000,E1 168.105} C_DIS
LIN {X -0.079,Y -372.104,Z 1407.727,A 0.000,B 0.000,C 90.000,E1 166.825} C_DIS
LIN {X 0.200,Y -385.414,Z 1407.719,A 0.000,B 0.000,C 90.000,E1 165.283} C_DIS
LIN {X -0.182,Y -397.631,Z 1407.712,A 0.000,B 0.000,C 90.000,E1 164.102} C_DIS
LIN {X -0.142,Y -411.585,Z 1407.705,A 0.000,B 0.000,C 90.000,E1 162.834} C_DIS
LIN {X 0.086,Y -427.089,Z 1407.697,A 0.000,B 0.000,C 90.000,E1 161.511} C_DIS
LIN {X 0.074,Y -439.713,Z 1407.692,A 0.000,B 0.000,C 90.000,E1 160.496} C_DIS
LIN {X 0.043,Y -450.446,Z 1407.687,A 0.000,B 0.000,C 90.000,E1 159.625} C_DIS
LIN {X -0.130,Y -459.463,Z 1407.683,A 0.000,B 0.000,C 90.000,E1 158.901} C_DIS
LIN {X 0.244,Y -469.830,Z 1407.678,A 0.000,B 0.000,C 90.000,E1 157.975} C_DIS
LIN {X -0.060,Y -480.093,Z 1407.673,A 0.000,B 0.000,C 90.000,E1 157.102} C_DIS
LIN {X -0.040,Y -488.746,Z 1407.668,A 0.000,B 0.000,C 90.000,E1 156.305} C_DIS
LIN {X 0.084,Y -497.163,Z 1407.664,A 0.000,B 0.000,C 90.000,E1 155.485} C_DIS
LIN {X -0.243,Y -502.531,Z 1407.661,A 0.000,B 0.000,C 90.000,E1 154.973} C_DIS
LIN {X 0.015,Y -509.124,Z 1407.657,A 0.000,B 0.000,C 90.000,E1 154.229} C_DIS
LIN {X 0.067,Y -514.193,Z 1407.654,A 0.000,B 0.000,C 90.000,E1 153.640} C_DIS
LIN {X 0.070,Y -518.993,Z 1407.650,A 0.000,B 0.000,C 90.000,E1 153.050} C_DIS
LIN {X -0.129,Y -523.388,Z 1407.647,A 0.000,B 0.000,C 90.000,E1 152.487} C_DIS
LIN {X 0.100,Y -526.491,Z 1407.645,A 0.000,B 0.000,C 90.000,E1 152.025} C_DIS
LIN {X 0.199,Y -530.171,Z 1407.641,A 0.000,B 0.000,C 90.000,E1 151.435} C_DIS
LIN {X 0.067,Y -533.401,Z 1407.638,A 0.000,B 0.000,C 90.000,E1 150.873} C_DIS
LIN {X 0.338,Y -536.861,Z 1407.634,A 0.000,B 0.000,C 90.000,E1 150.127} C_DIS
LIN {X 0.048,Y -539.278,Z 1407.631,A 0.000,B 0.000,C 90.000,E1 149.587} C_DIS
LIN {X -0.033,Y -542.386,Z 1407.626,A 0.000,B 0.000,C 90.000,E1 148.742} C_DIS
LIN {X -0.289,Y -544.255,Z 1407.623,A 0.000,B 0.000,C 90.000,E1 148.201} C_DIS
LIN {X 0.222,Y -545.955,Z 1407.620,A 0.000,B 0.000,C 90.000,E1 147.582} C_DIS
LIN {X 0.030,Y -548.176,Z 1407.615,A 0.000,B 0.000,C 90.000,E1 146.755} C_DIS
LIN {X -0.135,Y -550.031,Z 1407.611,A 0.000,B 0.000,C 90.000,E1 145.928} C_DIS
LIN {X 0.114,Y -551.139,Z 1407.608,A 0.000,B 0.000,C 90.000,E1 145.341} C_DIS
LIN {X 0.227,Y -552.125,Z 1407.604,A 0.000,B 0.000,C 90.000,E1 144.769} C_DIS
LIN {X -0.356,Y -553.244,Z 1407.600,A 0.000,B 0.000,C 90.000,E1 143.989} C_DIS
LIN {X -0.082,Y -554.440,Z 1407.594,A 0.000,B 0.000,C 90.000,E1 142.844} C_DIS
LIN {X -0.154,Y -555.689,Z 1407.586,A 0.000,B 0.000,C 90.000,E1 141.457} C_DIS
LIN {X -0.207,Y -556.927,Z 1407.578,A 0.000,B 0.000,C 90.000,E1 140.070} C_DIS
LIN {X -0.040,Y -557.520,Z 1407.573,A 0.000,B 0.000,C 90.000,E1 139.218} C_DIS
LIN {X 0.215,Y -558.184,Z 1407.567,A 0.000,B 0.000,C 90.000,E1 138.081} C_DIS
LIN {X 0.134,Y -558.898,Z 1407.560,A 0.000,B 0.000,C 90.000,E1 136.701} C_DIS
LIN {X -0.290,Y -559.519,Z 1407.550,A 0.000,B 0.000,C 90.000,E1 135.081} C_DIS
LIN {X 0.037,Y -559.941,Z 1407.543,A 0.000,B 0.000,C 90.000,E1 133.662} C_DIS
LIN {X -0.041,Y -560.229,Z 1407.535,A 0.000,B 0.000,C 90.000,E1 132.285} C_DIS
LIN {X 0.089,Y -560.371,Z 1407.524,A 0.000,B 0.000,C 90.000,E1 130.334} C_DIS
LIN {X 0.225,Y -560.676,Z 1407.513,A 0.000,B 0.000,C 90.000,E1 128.382} C_DIS
LIN {X -0.179,Y -560.828,Z 1407.507,A 0.000,B 0.000,C 90.000,E1 127.317} C_DIS
LIN {X -0.148,Y -560.847,Z 1407.500,A 0.000,B 0.000,C 90.000,E1 125.931} C_DIS
LIN {X -0.129,Y -560.910,Z 1407.489,A 0.000,B 0.000,C 90.000,E1 123.992} C_DIS
LIN {X -0.111,Y -561.254,Z 1407.478,A 0.000,B 0.000,C 90.000,E1 122.054} C_DIS
LIN {X 0.036,Y -562.061,Z 1407.474,A 0.000,B 0.000,C 90.000,E1 121.209} C_DIS
LIN {X -0.066,Y -562.269,Z 1407.473,A 0.000,B 0.000,C 90.000,E1 121.082} C_DIS
LIN {X -0.290,Y -563.469,Z 1407.471,A 0.000,B 0.000,C 90.000,E1 120.797} C_DIS
LIN {X -0.077,Y -563.976,Z 1407.469,A 0.000,B 0.000,C 90.000,E1 120.512} C_DIS
LIN {X -0.120,Y -564.033,Z 1407.469,A 0.000,B 0.000,C 90.000,E1 120.512} C_DIS
LIN {X 0.007,Y -565.680,Z 1407.469,A 0.000,B 0.000,C 90.000,E1 120.384} C_DIS
LIN {X -0.030,Y -567.014,Z 1407.469,A 0.000,B 0.000,C 90.000,E1 120.335} C_DIS
LIN {X 0.221,Y -570.653,Z 1407.468,A 0.000,B 0.000,C 90.000,E1 120.207} C_DIS
LIN {X -0.125,Y -576.922,Z 1407.467,A 0.000,B 0.000,C 90.000,E1 120.129} C_DIS
LIN {X 0.133,Y -582.378,Z 1407.467,A 0.000,B 0.000,C 90.000,E1 119.951} C_DIS
LIN {X -0.147,Y -585.241,Z 1407.466,A 0.000,B 0.000,C 90.000,E1 119.873} C_DIS
LIN {X -0.231,Y -589.232,Z 1407.465,A 0.000,B 0.000,C 90.000,E1 119.667} C_DIS
LIN {X 0.195,Y -590.678,Z 1407.464,A 0.000,B 0.000,C 90.000,E1 119.539} C_DIS
LIN {X -0.037,Y -595.995,Z 1407.462,A 0.000,B 0.000,C 90.000,E1 119.155} C_DIS
LIN {X -0.054,Y -601.204,Z 1407.459,A 0.000,B 0.000,C 90.000,E1 118.693} C_DIS
LIN {X 0.131,Y -605.123,Z 1407.457,A 0.000,B 0.000,C 90.000,E1 118.309} C_DIS
LIN {X 0.378,Y -609.837,Z 1407.454,A 0.000,B 0.000,C 90.000,E1 117.641} C_DIS
LIN {X 0.317,Y -612.401,Z 1407.452,A 0.000,B 0.000,C 90.000,E1 117.257} C_DIS
LIN {X 0.299,Y -613.149,Z 1407.451,A 0.000,B 0.000,C 90.000,E1 117.129} C_DIS
LIN {X 0.215,Y -615.939,Z 1407.447,A 0.000,B 0.000,C 90.000,E1 116.360} C_DIS
LIN {X 0.172,Y -616.375,Z 1407.444,A 0.000,B 0.000,C 90.000,E1 115.848} C_DIS
LIN {X 0.154,Y -616.430,Z 1407.442,A 0.000,B 0.000,C 90.000,E1 115.591} C_DIS
LIN {X 0.114,Y -615.135,Z 1407.439,A 0.000,B 0.000,C 90.000,E1 115.079} C_DIS
LIN {X 0.104,Y -614.718,Z 1407.439,A 0.000,B 0.000,C 90.000,E1 114.951} C_DIS
LIN {X -0.204,Y -611.314,Z 1407.436,A 0.000,B 0.000,C 90.000,E1 114.463} C_DIS
LIN {X -0.218,Y -609.982,Z 1407.435,A 0.000,B 0.000,C 90.000,E1 114.335} C_DIS
LIN {X -0.143,Y -607.027,Z 1407.434,A 0.000,B 0.000,C 90.000,E1 114.079} C_DIS
LIN {X -0.064,Y -605.163,Z 1407.433,A 0.000,B 0.000,C 90.000,E1 113.898} C_DIS
LIN {X 0.171,Y -597.312,Z 1407.431,A 0.000,B 0.000,C 90.000,E1 113.462} C_DIS
LIN {X -0.272,Y -582.516,Z 1407.427,A 0.000,B 0.000,C 90.000,E1 112.898} C_DIS
LIN {X 0.172,Y -582.158,Z 1407.427,A 0.000,B 0.000,C 90.000,E1 112.823} C_DIS
LIN {X 0.127,Y -582.203,Z 1407.427,A 0.000,B 0.000,C 90.000,E1 112.823} C_DIS
LIN {X -0.099,Y -584.077,Z 1407.426,A 0.000,B 0.000,C 90.000,E1 112.642} C_DIS
LIN {X -0.229,Y -584.901,Z 1407.425,A 0.000,B 0.000,C 90.000,E1 112.589} C_DIS
LIN {X 0.213,Y -590.685,Z 1407.424,A 0.000,B 0.000,C 90.000,E1 112.206} C_DIS
LIN {X -0.093,Y -595.156,Z 1407.422,A 0.000,B 0.000,C 90.000,E1 111.950} C_DIS
LIN {X -0.020,Y -600.962,Z 1407.420,A 0.000,B 0.000,C 90.000,E1 111.535} C_DIS
LIN {X 0.109,Y -606.385,Z 1407.417,A 0.000,B 0.000,C 90.000,E1 111.099} C_DIS
LIN {X -0.267,Y -610.407,Z 1407.415,A 0.000,B 0.000,C 90.000,E1 110.791} C_DIS
LIN {X 0.129,Y -617.675,Z 1407.412,A 0.000,B 0.000,C 90.000,E1 110.066} C_DIS
LIN {X 0.184,Y -620.076,Z 1407.410,A 0.000,B 0.000,C 90.000,E1 109.812} C_DIS
LIN {X -0.276,Y -625.653,Z 1407.407,A 0.000,B 0.000,C 90.000,E1 109.214} C_DIS
LIN {X 0.090,Y -630.388,Z 1407.403,A 0.000,B 0.000,C 90.000,E1 108.544} C_DIS
LIN {X -0.109,Y -633.832,Z 1407.400,A 0.000,B 0.000,C 90.000,E1 108.055} C_DIS
LIN {X 0.316,Y -636.855,Z 1407.397,A 0.000,B 0.000,C 90.000,E1 107.511} C_DIS
LIN {X -0.044,Y -638.776,Z 1407.395,A 0.000,B 0.000,C 90.000,E1 107.166} C_DIS
LIN {X -0.027,Y -639.943,Z 1407.394,A 0.000,B 0.000,C 90.000,E1 106.913} C_DIS
LIN {X 0.254,Y -641.876,Z 1407.391,A 0.000,B 0.000,C 90.000,E1 106.386} C_DIS
LIN {X 0.096,Y -642.703,Z 1407.390,A 0.000,B 0.000,C 90.000,E1 106.150} C_DIS
LIN {X -0.192,Y -644.238,Z 1407.386,A 0.000,B 0.000,C 90.000,E1 105.426} C_DIS
LIN {X 0.132,Y -645.067,Z 1407.383,A 0.000,B 0.000,C 90.000,E1 104.898} C_DIS
LIN {X 0.195,Y -646.632,Z 1407.376,A 0.000,B 0.000,C 90.000,E1 103.647} C_DIS
LIN {X -0.090,Y -647.052,Z 1407.373,A 0.000,B 0.000,C 90.000,E1 103.175} C_DIS
LIN {X 0.117,Y -647.219,Z 1407.369,A 0.000,B 0.000,C 90.000,E1 102.411} C_DIS
LIN {X -0.301,Y -647.085,Z 1407.366,A 0.000,B 0.000,C 90.000,E1 101.951} C_DIS
LIN {X 0.051,Y -646.777,Z 1407.364,A 0.000,B 0.000,C 90.000,E1 101.422} C_DIS
LIN {X -0.236,Y -646.232,Z 1407.361,A 0.000,B 0.000,C 90.000,E1 100.950} C_DIS
LIN {X -0.160,Y -645.006,Z 1407.357,A 0.000,B 0.000,C 90.000,E1 100.197} C_DIS
LIN {X 0.171,Y -643.911,Z 1407.354,A 0.000,B 0.000,C 90.000,E1 99.670} C_DIS
LIN {X -0.249,Y -642.547,Z 1407.351,A 0.000,B 0.000,C 90.000,E1 99.208} C_DIS
LIN {X 0.060,Y -640.963,Z 1407.348,A 0.000,B 0.000,C 90.000,E1 98.681} C_DIS
LIN {X 0.258,Y -639.182,Z 1407.346,A 0.000,B 0.000,C 90.000,E1 98.163} C_DIS
LIN {X -0.184,Y -637.106,Z 1407.343,A 0.000,B 0.000,C 90.000,E1 97.701} C_DIS
LIN {X -0.199,Y -633.670,Z 1407.339,A 0.000,B 0.000,C 90.000,E1 96.947} C_DIS
LIN {X -0.188,Y -630.359,Z 1407.335,A 0.000,B 0.000,C 90.000,E1 96.315} C_DIS
LIN {X 0.194,Y -625.302,Z 1407.330,A 0.000,B 0.000,C 90.000,E1 95.391} C_DIS
LIN {X 0.132,Y -621.132,Z 1407.327,A 0.000,B 0.000,C 90.000,E1 94.759} C_DIS
LIN {X 0.143,Y -617.222,Z 1407.324,A 0.000,B 0.000,C 90.000,E1 94.245} C_DIS
LIN {X -0.122,Y -614.933,Z 1407.322,A 0.000,B 0.000,C 90.000,E1 94.012} C_DIS
LIN {X 0.103,Y -610.061,Z 1407.320,A 0.000,B 0.000,C 90.000,E1 93.498} C_DIS
LIN {X -0.056,Y -603.405,Z 1407.316,A 0.000,B 0.000,C 90.000,E1 92.922} C_DIS
LIN {X -0.164,Y -596.528,Z 1407.313,A 0.000,B 0.000,C 90.000,E1 92.350} C_DIS
LIN {X 0.059,Y -590.908,Z 1407.311,A 0.000,B 0.000,C 90.000,E1 91.892} C_DIS
LIN {X 0.228,Y -587.585,Z 1407.309,A 0.000,B 0.000,C 90.000,E1 91.661} C_DIS
LIN {X -0.191,Y -580.923,Z 1407.307,A 0.000,B 0.000,C 90.000,E1 91.318} C_DIS
LIN {X -0.267,Y -577.608,Z 1407.306,A 0.000,B 0.000,C 90.000,E1 91.146} C_DIS
LIN {X -0.061,Y -574.048,Z 1407.304,A 0.000,B 0.000,C 90.000,E1 90.802} C_DIS
LIN {X -0.100,Y -574.000,Z 1407.304,A 0.000,B 0.000,C 90.000,E1 90.802} C_DIS
LIN {X -0.227,Y -573.234,Z 1407.303,A 0.000,B 0.000,C 90.000,E1 90.573} C_DIS
LIN {X 0.274,Y -573.028,Z 1407.301,A 0.000,B 0.000,C 90.000,E1 90.115} C_DIS
LIN {X 0.126,Y -573.492,Z 1407.296,A 0.000,B 0.000,C 90.000,E1 89.312} C_DIS
LIN {X 0.288,Y -574.768,Z 1407.289,A 0.000,B 0.000,C 90.000,E1 87.936} C_DIS
LIN {X 0.047,Y -576.219,Z 1407.280,A 0.000,B 0.000,C 90.000,E1 86.331} C_DIS
LIN {X 0.210,Y -578.368,Z 1407.268,A 0.000,B 0.000,C 90.000,E1 84.147} C_DIS
LIN {X -0.021,Y -579.899,Z 1407.260,A 0.000,B 0.000,C 90.000,E1 82.818} C_DIS
LIN {X 0.232,Y -582.086,Z 1407.250,A 0.000,B 0.000,C 90.000,E1 80.905} C_DIS
LIN {X -0.282,Y -583.924,Z 1407.241,A 0.000,B 0.000,C 90.000,E1 79.342} C_DIS
LIN {X -0.220,Y -585.288,Z 1407.233,A 0.000,B 0.000,C 90.000,E1 77.993} C_DIS
LIN {X 0.192,Y -586.182,Z 1407.227,A 0.000,B 0.000,C 90.000,E1 76.881} C_DIS
LIN {X -0.137,Y -587.296,Z 1407.220,A 0.000,B 0.000,C 90.000,E1 75.574} C_DIS
LIN {X 0.127,Y -588.181,Z 1407.212,A 0.000,B 0.000,C 90.000,E1 74.212} C_DIS
LIN {X 0.249,Y -589.051,Z 1407.203,A 0.000,B 0.000,C 90.000,E1 72.598} C_DIS
LIN {X 0.139,Y -589.818,Z 1407.196,A 0.000,B 0.000,C 90.000,E1 71.275} C_DIS
LIN {X -0.210,Y -590.843,Z 1407.186,A 0.000,B 0.000,C 90.000,E1 69.444} C_DIS
LIN {X 0.227,Y -591.961,Z 1407.175,A 0.000,B 0.000,C 90.000,E1 67.539} C_DIS
LIN {X 0.370,Y -593.233,Z 1407.165,A 0.000,B 0.000,C 90.000,E1 65.665} C_DIS
LIN {X -0.008,Y -594.691,Z 1407.155,A 0.000,B 0.000,C 90.000,E1 63.845} C_DIS
LIN {X -0.187,Y -595.754,Z 1407.147,A 0.000,B 0.000,C 90.000,E1 62.538} C_DIS
LIN {X 0.103,Y -597.032,Z 1407.139,A 0.000,B 0.000,C 90.000,E1 60.923} C_DIS
LIN {X 0.055,Y -598.023,Z 1407.133,A 0.000,B 0.000,C 90.000,E1 59.871} C_DIS
LIN {X -0.128,Y -599.718,Z 1407.122,A 0.000,B 0.000,C 90.000,E1 58.043} C_DIS
LIN {X 0.083,Y -600.915,Z 1407.115,A 0.000,B 0.000,C 90.000,E1 56.707} C_DIS
LIN {X -0.202,Y -602.602,Z 1407.105,A 0.000,B 0.000,C 90.000,E1 54.895} C_DIS
LIN {X 0.131,Y -603.987,Z 1407.096,A 0.000,B 0.000,C 90.000,E1 53.290} C_DIS
LIN {X 0.101,Y -604.933,Z 1407.089,A 0.000,B 0.000,C 90.000,E1 51.984} C_DIS
LIN {X -0.176,Y -605.655,Z 1407.083,A 0.000,B 0.000,C 90.000,E1 50.964} C_DIS
LIN {X 0.202,Y -606.360,Z 1407.076,A 0.000,B 0.000,C 90.000,E1 49.622} C_DIS
LIN {X 0.067,Y -606.648,Z 1407.072,A 0.000,B 0.000,C 90.000,E1 48.852} C_DIS
LIN {X 0.196,Y -606.891,Z 1407.066,A 0.000,B 0.000,C 90.000,E1 47.796} C_DIS
LIN {X 0.163,Y -607.043,Z 1407.056,A 0.000,B 0.000,C 90.000,E1 45.972} C_DIS
LIN {X 0.080,Y -606.897,Z 1407.048,A 0.000,B 0.000,C 90.000,E1 44.676} C_DIS
LIN {X 0.180,Y -606.559,Z 1407.042,A 0.000,B 0.000,C 90.000,E1 43.623} C_DIS
LIN {X -0.143,Y -606.084,Z 1407.037,A 0.000,B 0.000,C 90.000,E1 42.609} C_DIS
LIN {X -0.022,Y -605.490,Z 1407.031,A 0.000,B 0.000,C 90.000,E1 41.553} C_DIS
LIN {X -0.361,Y -604.685,Z 1407.025,A 0.000,B 0.000,C 90.000,E1 40.539} C_DIS
LIN {X -0.260,Y -603.757,Z 1407.019,A 0.000,B 0.000,C 90.000,E1 39.483} C_DIS
LIN {X -0.299,Y -602.313,Z 1407.012,A 0.000,B 0.000,C 90.000,E1 38.177} C_DIS
LIN {X 0.232,Y -600.903,Z 1407.006,A 0.000,B 0.000,C 90.000,E1 37.076} C_DIS
LIN {X 0.132,Y -599.730,Z 1407.002,A 0.000,B 0.000,C 90.000,E1 36.297} C_DIS
LIN {X 0.152,Y -597.322,Z 1406.995,A 0.000,B 0.000,C 90.000,E1 34.978} C_DIS
LIN {X 0.018,Y -595.609,Z 1406.990,A 0.000,B 0.000,C 90.000,E1 34.199} C_DIS
LIN {X -0.250,Y -593.108,Z 1406.984,A 0.000,B 0.000,C 90.000,E1 33.166} C_DIS
LIN {X -0.053,Y -590.214,Z 1406.978,A 0.000,B 0.000,C 90.000,E1 32.084} C_DIS
LIN {X 0.221,Y -587.773,Z 1406.974,A 0.000,B 0.000,C 90.000,E1 31.258} C_DIS
LIN {X 0.160,Y -584.957,Z 1406.969,A 0.000,B 0.000,C 90.000,E1 30.463} C_DIS
LIN {X 0.201,Y -582.856,Z 1406.966,A 0.000,B 0.000,C 90.000,E1 29.922} C_DIS
LIN {X -0.196,Y -579.273,Z 1406.962,A 0.000,B 0.000,C 90.000,E1 29.155} C_DIS
LIN {X 0.160,Y -575.435,Z 1406.957,A 0.000,B 0.000,C 90.000,E1 28.309} C_DIS
LIN {X -0.286,Y -568.874,Z 1406.951,A 0.000,B 0.000,C 90.000,E1 27.129} C_DIS
LIN {X 0.263,Y -562.451,Z 1406.944,A 0.000,B 0.000,C 90.000,E1 25.976} C_DIS
LIN {X 0.072,Y -556.194,Z 1406.939,A 0.000,B 0.000,C 90.000,E1 25.027} C_DIS
LIN {X -0.079,Y -550.280,Z 1406.934,A 0.000,B 0.000,C 90.000,E1 24.207} C_DIS
LIN {X 0.071,Y -547.123,Z 1406.932,A 0.000,B 0.000,C 90.000,E1 23.770} C_DIS
LIN {X -0.048,Y -541.545,Z 1406.928,A 0.000,B 0.000,C 90.000,E1 23.078} C_DIS
LIN {X -0.080,Y -536.836,Z 1406.925,A 0.000,B 0.000,C 90.000,E1 22.514} C_DIS
LIN {X -0.132,Y -529.330,Z 1406.920,A 0.000,B 0.000,C 90.000,E1 21.663} C_DIS
LIN {X -0.231,Y -524.136,Z 1406.917,A 0.000,B 0.000,C 90.000,E1 21.099} C_DIS
LIN {X -0.167,Y -515.111,Z 1406.912,A 0.000,B 0.000,C 90.000,E1 20.120} C_DIS
LIN {X 0.007,Y -504.731,Z 1406.906,A 0.000,B 0.000,C 90.000,E1 19.033} C_DIS
LIN {X -0.106,Y -492.702,Z 1406.899,A 0.000,B 0.000,C 90.000,E1 17.819} C_DIS
LIN {X -0.008,Y -477.789,Z 1406.890,A 0.000,B 0.000,C 90.000,E1 16.260} C_DIS
LIN {X 0.005,Y -462.904,Z 1406.881,A 0.000,B 0.000,C 90.000,E1 14.662} C_DIS
LIN {X -0.131,Y -449.140,Z 1406.873,A 0.000,B 0.000,C 90.000,E1 13.175} C_DIS
LIN {X -0.172,Y -433.971,Z 1406.864,A 0.000,B 0.000,C 90.000,E1 11.478} C_DIS
LIN {X -0.130,Y -413.854,Z 1406.850,A 0.000,B 0.000,C 90.000,E1 9.029} C_DIS
LIN {X -0.060,Y -403.256,Z 1406.843,A 0.000,B 0.000,C 90.000,E1 7.644} C_DIS
LIN {X 0.005,Y -396.642,Z 1406.838,A 0.000,B 0.000,C 90.000,E1 6.777} C_DIS
LIN {X -0.037,Y -392.711,Z 1406.835,A 0.000,B 0.000,C 90.000,E1 6.258} C_DIS
LIN {X 0.195,Y -389.550,Z 1406.832,A 0.000,B 0.000,C 90.000,E1 5.739} C_DIS
LIN {X 0.152,Y -388.595,Z 1406.831,A 0.000,B 0.000,C 90.000,E1 5.568} C_DIS
LIN {X -0.065,Y -387.195,Z 1406.829,A 0.000,B 0.000,C 90.000,E1 5.277} C_DIS
LIN {X -0.103,Y -387.174,Z 1406.829,A 0.000,B 0.000,C 90.000,E1 5.277} C_DIS
LIN {X 0.057,Y -387.174,Z 1406.829,A 0.000,B 0.000,C 90.000,E1 5.220} C_DIS
LIN {X 0.019,Y -387.180,Z 1406.829,A 0.000,B 0.000,C 90.000,E1 5.220} C_DIS
LIN {X 0.060,Y -388.676,Z 1406.828,A 0.000,B 0.000,C 90.000,E1 4.935} C_DIS
LIN {X -0.163,Y -392.391,Z 1406.825,A 0.000,B 0.000,C 90.000,E1 4.531} C_DIS
LIN {X -0.060,Y -400.965,Z 1406.820,A 0.000,B 0.000,C 90.000,E1 3.669} C_DIS
LIN {X -0.074,Y -405.261,Z 1406.818,A 0.000,B 0.000,C 90.000,E1 3.212} C_DIS
LIN {X 0.109,Y -410.294,Z 1406.814,A 0.000,B 0.000,C 90.000,E1 2.522} C_DIS
LIN {X 0.097,Y -415.119,Z 1406.810,A 0.000,B 0.000,C 90.000,E1 1.835} C_DIS
LIN {X 0.148,Y -420.036,Z 1406.806,A 0.000,B 0.000,C 90.000,E1 0.974} C_DIS
LIN {X 0.196,Y -422.604,Z 1406.803,A 0.000,B 0.000,C 90.000,E1 0.458} C_DIS
LIN {X 0.000,Y -424.699,Z 1406.800,A 0.000,B 0.000,C 90.000,E1 360.000} C_DIS
LIN {X 0.161,Y -425.460,Z 1406.799,A 0.000,B 0.000,C 90.000,E1 359.771} C_DIS
LIN {X -0.212,Y -426.367,Z 1406.797,A 0.000,B 0.000,C 90.000,E1 359.484} C_DIS
LIN {X -0.157,Y -426.610,Z 1406.795,A 0.000,B 0.000,C 90.000,E1 359.141} C_DIS
LIN {X 0.094,Y -426.284,Z 1406.794,A 0.000,B 0.000,C 90.000,E1 358.969} C_DIS
LIN {X -0.213,Y -425.581,Z 1406.794,A 0.000,B 0.000,C 90.000,E1 358.912} C_DIS
LIN {X -0.080,Y -424.901,Z 1406.794,A 0.000,B 0.000,C 90.000,E1 358.854} C_DIS
LIN {X -0.190,Y -424.289,Z 1406.794,A 0.000,B 0.000,C 90.000,E1 358.854} C_DIS
LIN {X 0.009,Y -361.234,Z 1406.792,A 0.000,B 0.000,C 90.000,E1 358.625} C_DIS
LIN {X -0.020,Y -360.134,Z 1406.792,A 0.000,B 0.000,C 90.000,E1 358.625} C_DIS
LIN {X 0.067,Y -359.402,Z 1406.768,A 0.000,B 0.000,C 90.000,E1 354.261} C_DIS
LIN {X -0.031,Y -359.514,Z 1406.726,A 0.000,B 0.000,C 90.000,E1 346.756} C_DIS
LIN {X -0.126,Y -359.528,Z 1406.720,A 0.000,B 0.000,C 90.000,E1 345.644} C_DIS
LIN {X -0.192,Y -361.968,Z 1406.683,A 0.000,B 0.000,C 90.000,E1 338.901} C_DIS
LIN {X 0.064,Y -365.874,Z 1406.643,A 0.000,B 0.000,C 90.000,E1 331.769} C_DIS
LIN {X 0.143,Y -366.199,Z 1406.641,A 0.000,B 0.000,C 90.000,E1 331.385} C_DIS
LIN {X -0.154,Y -371.230,Z 1406.604,A 0.000,B 0.000,C 90.000,E1 324.769} C_DIS
LIN {X -0.167,Y -371.664,Z 1406.602,A 0.000,B 0.000,C 90.000,E1 324.402} C_DIS
LIN {X -0.111,Y -376.769,Z 1406.570,A 0.000,B 0.000,C 90.000,E1 318.528} C_DIS
LIN {X 0.179,Y -378.159,Z 1406.563,A 0.000,B 0.000,C 90.000,E1 317.391} C_DIS
LIN {X 0.165,Y -383.798,Z 1406.531,A 0.000,B 0.000,C 90.000,E1 311.595} C_DIS
LIN {X -0.040,Y -384.790,Z 1406.527,A 0.000,B 0.000,C 90.000,E1 310.906} C_DIS
LIN {X -0.050,Y -390.959,Z 1406.493,A 0.000,B 0.000,C 90.000,E1 304.818} C_DIS
LIN {X 0.016,Y -391.368,Z 1406.491,A 0.000,B 0.000,C 90.000,E1 304.452} C_DIS
LIN {X -0.254,Y -396.690,Z 1406.460,A 0.000,B 0.000,C 90.000,E1 298.821} C_DIS
LIN {X -0.035,Y -397.075,Z 1406.458,A 0.000,B 0.000,C 90.000,E1 298.437} C_DIS
LIN {X -0.080,Y -401.491,Z 1406.427,A 0.000,B 0.000,C 90.000,E1 292.823} C_DIS
LIN {X 0.087,Y -401.769,Z 1406.423,A 0.000,B 0.000,C 90.000,E1 292.099} C_DIS
LIN {X 0.046,Y -404.568,Z 1406.396,A 0.000,B 0.000,C 90.000,E1 287.221} C_DIS
LIN {X 0.148,Y -404.760,Z 1406.394,A 0.000,B 0.000,C 90.000,E1 286.858} C_DIS
LIN {X 0.055,Y -406.041,Z 1406.365,A 0.000,B 0.000,C 90.000,E1 281.658} C_DIS
LIN {X 0.145,Y -406.137,Z 1406.363,A 0.000,B 0.000,C 90.000,E1 281.299} C_DIS
LIN {X 0.175,Y -405.656,Z 1406.334,A 0.000,B 0.000,C 90.000,E1 276.087} C_DIS
LIN {X 0.180,Y -405.599,Z 1406.332,A 0.000,B 0.000,C 90.000,E1 275.739} C_DIS
LIN {X -0.150,Y -403.548,Z 1406.305,A 0.000,B 0.000,C 90.000,E1 270.917} C_DIS
LIN {X 0.188,Y -403.037,Z 1406.301,A 0.000,B 0.000,C 90.000,E1 270.172} C_DIS
LIN {X 0.010,Y -399.008,Z 1406.272,A 0.000,B 0.000,C 90.000,E1 264.951} C_DIS
LIN {X -0.191,Y -396.730,Z 1406.262,A 0.000,B 0.000,C 90.000,E1 263.223} C_DIS
LIN {X -0.215,Y -392.921,Z 1406.241,A 0.000,B 0.000,C 90.000,E1 259.342} C_DIS
LIN {X 0.161,Y -391.864,Z 1406.237,A 0.000,B 0.000,C 90.000,E1 258.578} C_DIS
LIN {X -0.084,Y -385.728,Z 1406.211,A 0.000,B 0.000,C 90.000,E1 253.976} C_DIS
LIN {X -0.148,Y -384.961,Z 1406.207,A 0.000,B 0.000,C 90.000,E1 253.268} C_DIS
LIN {X 0.080,Y -378.109,Z 1406.183,A 0.000,B 0.000,C 90.000,E1 248.901} C_DIS
LIN {X -0.185,Y -376.351,Z 1406.175,A 0.000,B 0.000,C 90.000,E1 247.486} C_DIS
LIN {X -0.060,Y -375.846,Z 1406.173,A 0.000,B 0.000,C 90.000,E1 247.102} C_DIS
LIN {X 0.059,Y -369.078,Z 1406.150,A 0.000,B 0.000,C 90.000,E1 243.050} C_DIS
LIN {X -0.030,Y -366.231,Z 1406.138,A 0.000,B 0.000,C 90.000,E1 240.845} C_DIS
LIN {X -0.068,Y -358.826,Z 1406.113,A 0.000,B 0.000,C 90.000,E1 236.373} C_DIS
LIN {X -0.079,Y -356.017,Z 1406.101,A 0.000,B 0.000,C 90.000,E1 234.116} C_DIS
LIN {X -0.082,Y -348.455,Z 1406.073,A 0.000,B 0.000,C 90.000,E1 229.175} C_DIS
LIN {X -0.021,Y -345.867,Z 1406.060,A 0.000,B 0.000,C 90.000,E1 226.863} C_DIS
LIN {X -0.054,Y -339.102,Z 1406.032,A 0.000,B 0.000,C 90.000,E1 221.838} C_DIS
LIN {X 0.031,Y -336.942,Z 1406.019,A 0.000,B 0.000,C 90.000,E1 219.483} C_DIS
LIN {X 0.010,Y -331.617,Z 1405.993,A 0.000,B 0.000,C 90.000,E1 214.771} C_DIS
LIN {X 0.082,Y -329.358,Z 1405.976,A 0.000,B 0.000,C 90.000,E1 211.592} C_DIS
LIN {X 0.093,Y -328.627,Z 1405.971,A 0.000,B 0.000,C 90.000,E1 210.797} C_DIS
LIN {X 0.007,Y -324.086,Z 1405.934,A 0.000,B 0.000,C 90.000,E1 204.027} C_DIS
LIN {X 0.112,Y -323.865,Z 1405.929,A 0.000,B 0.000,C 90.000,E1 203.206} C_DIS
LIN {X 0.184,Y -322.853,Z 1405.920,A 0.000,B 0.000,C 90.000,E1 201.589} C_DIS
LIN {X 0.098,Y -321.117,Z 1405.880,A 0.000,B 0.000,C 90.000,E1 194.356} C_DIS
LIN {X -0.054,Y -321.506,Z 1405.833,A 0.000,B 0.000,C 90.000,E1 185.910} C_DIS
LIN {X -0.056,Y -321.639,Z 1405.826,A 0.000,B 0.000,C 90.000,E1 184.702} C_DIS
LIN {X 0.156,Y -322.215,Z 1405.812,A 0.000,B 0.000,C 90.000,E1 182.064} C_DIS
LIN {X 0.128,Y -322.671,Z 1405.812,A 0.000,B 0.000,C 90.000,E1 182.064} C_DIS
LIN {X -0.128,Y -398.414,Z 1405.809,A 0.000,B 0.000,C 90.000,E1 181.718} C_DIS
LIN {X 0.144,Y -399.361,Z 1405.809,A 0.000,B 0.000,C 90.000,E1 181.661} C_DIS
LIN {X 0.032,Y -400.339,Z 1405.809,A 0.000,B 0.000,C 90.000,E1 181.604} C_DIS
LIN {X -0.082,Y -401.160,Z 1405.808,A 0.000,B 0.000,C 90.000,E1 181.375} C_DIS
LIN {X -0.128,Y -400.976,Z 1405.806,A 0.000,B 0.000,C 90.000,E1 181.031} C_DIS
LIN {X -0.170,Y -400.234,Z 1405.804,A 0.000,B 0.000,C 90.000,E1 180.688} C_DIS
LIN {X 0.186,Y -399.212,Z 1405.802,A 0.000,B 0.000,C 90.000,E1 180.286} C_DIS
LIN {X 0.063,Y -396.156,Z 1405.797,A 0.000,B 0.000,C 90.000,E1 179.427} C_DIS
LIN {X -0.130,Y -391.874,Z 1405.791,A 0.000,B 0.000,C 90.000,E1 178.396} C_DIS
LIN {X 0.070,Y -387.679,Z 1405.786,A 0.000,B 0.000,C 90.000,E1 177.478} C_DIS
LIN {X 0.171,Y -382.004,Z 1405.780,A 0.000,B 0.000,C 90.000,E1 176.388} C_DIS
LIN {X -0.112,Y -376.832,Z 1405.775,A 0.000,B 0.000,C 90.000,E1 175.527} C_DIS
LIN {X 0.083,Y -373.698,Z 1405.772,A 0.000,B 0.000,C 90.000,E1 174.951} C_DIS
LIN {X -0.047,Y -367.006,Z 1405.765,A 0.000,B 0.000,C 90.000,E1 173.685} C_DIS
LIN {X -0.028,Y -359.024,Z 1405.756,A 0.000,B 0.000,C 90.000,E1 172.008} C_DIS
LIN {X -0.133,Y -355.135,Z 1405.750,A 0.000,B 0.000,C 90.000,E1 171.084} C_DIS
LIN {X -0.030,Y -353.287,Z 1405.747,A 0.000,B 0.000,C 90.000,E1 170.500} C_DIS
LIN {X -0.015,Y -352.233,Z 1405.744,A 0.000,B 0.000,C 90.000,E1 169.982} C_DIS
LIN {X -0.034,Y -352.241,Z 1405.744,A 0.000,B 0.000,C 90.000,E1 169.982} C_DIS
LIN {X -0.063,Y -352.836,Z 1405.743,A 0.000,B 0.000,C 90.000,E1 169.746} C_DIS
LIN {X -0.057,Y -353.325,Z 1405.741,A 0.000,B 0.000,C 90.000,E1 169.454} C_DIS
LIN {X -0.076,Y -353.339,Z 1405.741,A 0.000,B 0.000,C 90.000,E1 169.454} C_DIS
LIN {X -0.168,Y -357.166,Z 1405.738,A 0.000,B 0.000,C 90.000,E1 168.814} C_DIS
LIN {X 0.128,Y -364.945,Z 1405.732,A 0.000,B 0.000,C 90.000,E1 167.701} C_DIS
LIN {X -0.025,Y -373.632,Z 1405.726,A 0.000,B 0.000,C 90.000,E1 166.645} C_DIS
LIN {X 0.166,Y -385.586,Z 1405.718,A 0.000,B 0.000,C 90.000,E1 165.283} C_DIS
LIN {X -0.219,Y -397.813,Z 1405.712,A 0.000,B 0.000,C 90.000,E1 164.102} C_DIS
LIN {X 0.068,Y -413.261,Z 1405.704,A 0.000,B 0.000,C 90.000,E1 162.670} C_DIS
LIN {X -0.169,Y -430.541,Z 1405.696,A 0.000,B 0.000,C 90.000,E1 161.275} C_DIS
LIN {X 0.007,Y -441.522,Z 1405.691,A 0.000,B 0.000,C 90.000,E1 160.369} C_DIS
LIN {X -0.240,Y -452.433,Z 1405.686,A 0.000,B 0.000,C 90.000,E1 159.518} C_DIS
LIN {X 0.064,Y -460.077,Z 1405.683,A 0.000,B 0.000,C 90.000,E1 158.847} C_DIS
LIN {X -0.142,Y -470.611,Z 1405.678,A 0.000,B 0.000,C 90.000,E1 157.975} C_DIS
LIN {X 0.047,Y -477.948,Z 1405.674,A 0.000,B 0.000,C 90.000,E1 157.305} C_DIS
LIN {X -0.180,Y -486.595,Z 1405.670,A 0.000,B 0.000,C 90.000,E1 156.538} C_DIS
LIN {X -0.052,Y -495.097,Z 1405.665,A 0.000,B 0.000,C 90.000,E1 155.717} C_DIS
LIN {X -0.101,Y -500.590,Z 1405.662,A 0.000,B 0.000,C 90.000,E1 155.177} C_DIS
LIN {X 0.110,Y -505.893,Z 1405.659,A 0.000,B 0.000,C 90.000,E1 154.588} C_DIS
LIN {X 0.108,Y -513.664,Z 1405.654,A 0.000,B 0.000,C 90.000,E1 153.717} C_DIS
LIN {X 0.214,Y -518.430,Z 1405.651,A 0.000,B 0.000,C 90.000,E1 153.127} C_DIS
LIN {X 0.010,Y -522.851,Z 1405.648,A 0.000,B 0.000,C 90.000,E1 152.564} C_DIS
LIN {X 0.077,Y -526.933,Z 1405.644,A 0.000,B 0.000,C 90.000,E1 151.975} C_DIS
LIN {X 0.176,Y -530.614,Z 1405.641,A 0.000,B 0.000,C 90.000,E1 151.385} C_DIS
LIN {X -0.162,Y -533.828,Z 1405.638,A 0.000,B 0.000,C 90.000,E1 150.845} C_DIS
LIN {X -0.151,Y -537.214,Z 1405.634,A 0.000,B 0.000,C 90.000,E1 150.127} C_DIS
LIN {X 0.026,Y -539.622,Z 1405.631,A 0.000,B 0.000,C 90.000,E1 149.537} C_DIS
